LIN {X 0,Y 532.094,Z 203.208,A -85,B 0,C 180,E1 -4182.718,E2 -4182.718} C_VEL
LIN {X 0,Y 531.047,Z 203.336,A -85,B 0,C 180,E1 -4183.349,E2 -4183.349} C_VEL
LIN {X 0,Y 530.959,Z 203.344,A -85,B 0,C 180,E1 -4183.563,E2 -4183.563} C_VEL
LIN {X 0,Y 530.963,Z 203.345,A -85,B 0,C 180,E1 -4186.507,E2 -4186.507} C_VEL
LIN {X 0,Y 530.986,Z 203.345,A -85,B 0,C 180,E1 -4188.977,E2 -4188.977} C_VEL
LIN {X 0,Y 530.955,Z 203.343,A -85,B 0,C 180,E1 -4191.53,E2 -4191.53} C_VEL
LIN {X 0,Y 530.953,Z 203.348,A -85,B 0,C 180,E1 -4194.381,E2 -4194.381} C_VEL
LIN {X 0,Y 531.017,Z 203.34,A -85,B 0,C 180,E1 -4197.138,E2 -4197.138} C_VEL
LIN {X 0,Y 530.961,Z 203.352,A -85,B 0,C 180,E1 -4198.311,E2 -4198.311} C_VEL
LIN {X 0,Y 530.989,Z 212.149,A -85,B 0,C 180,E1 -4199.578,E2 -4199.578} C_VEL
LIN {X 0,Y 531.066,Z 222.092,A -85,B 0,C 180,E1 -4201.078,E2 -4201.078} C_VEL
LIN {X 0,Y 532.836,Z 233.019,A -85,B 0,C 180,E1 -4201.293,E2 -4201.293} C_VEL
LIN {X 0,Y 532.369,Z 329.637,A -85,B 0,C 180,E1 -4202.615,E2 -4202.615} C_VEL
LIN {X 0,Y 532.211,Z 343.265,A -85,B 0,C 180,E1 -4202.952,E2 -4202.952} C_VEL
LIN {X 0,Y 532.009,Z 355.388,A -85,B 0,C 180,E1 -4203.408,E2 -4203.408} C_VEL
LIN {X 0,Y 531.839,Z 368.214,A -85,B 0,C 180,E1 -4204.069,E2 -4204.069} C_VEL
LIN {X 0,Y 531.531,Z 378.711,A -85,B 0,C 180,E1 -4204.761,E2 -4204.761} C_VEL
LIN {X 0,Y 531.349,Z 388.715,A -85,B 0,C 180,E1 -4205.587,E2 -4205.587} C_VEL
LIN {X 0,Y 531.056,Z 398.766,A -85,B 0,C 180,E1 -4206.609,E2 -4206.609} C_VEL
LIN {X 0,Y 530.884,Z 407.591,A -85,B 0,C 180,E1 -4207.727,E2 -4207.727} C_VEL
LIN {X 0,Y 530.71,Z 414.712,A -85,B 0,C 180,E1 -4208.848,E2 -4208.848} C_VEL
LIN {X 0,Y 530.596,Z 421.185,A -85,B 0,C 180,E1 -4210.125,E2 -4210.125} C_VEL
LIN {X 0,Y 530.511,Z 426.324,A -85,B 0,C 180,E1 -4211.462,E2 -4211.462} C_VEL
LIN {X 0,Y 530.462,Z 429.415,A -85,B 0,C 180,E1 -4212.54,E2 -4212.54} C_VEL
LIN {X 0,Y 530.377,Z 431.976,A -85,B 0,C 180,E1 -4213.844,E2 -4213.844} C_VEL
LIN {X 0,Y 530.394,Z 433.447,A -85,B 0,C 180,E1 -4215.307,E2 -4215.307} C_VEL
LIN {X 0,Y 530.393,Z 433.621,A -85,B 0,C 180,E1 -4216.202,E2 -4216.202} C_VEL
LIN {X 0,Y 530.39,Z 433.323,A -85,B 0,C 180,E1 -4216.983,E2 -4216.983} C_VEL
LIN {X 0,Y 530.405,Z 432.632,A -85,B 0,C 180,E1 -4217.761,E2 -4217.761} C_VEL
LIN {X 0,Y 530.452,Z 431.3,A -85,B 0,C 180,E1 -4218.649,E2 -4218.649} C_VEL
LIN {X 0,Y 530.506,Z 427.984,A -85,B 0,C 180,E1 -4220.084,E2 -4220.084} C_VEL
LIN {X 0,Y 530.552,Z 424.156,A -85,B 0,C 180,E1 -4221.239,E2 -4221.239} C_VEL
LIN {X 0,Y 530.628,Z 419.211,A -85,B 0,C 180,E1 -4222.39,E2 -4222.39} C_VEL
LIN {X 0,Y 530.755,Z 412.935,A -85,B 0,C 180,E1 -4223.544,E2 -4223.544} C_VEL
LIN {X 0,Y 530.896,Z 405.219,A -85,B 0,C 180,E1 -4224.684,E2 -4224.684} C_VEL
LIN {X 0,Y 531.086,Z 397.332,A -85,B 0,C 180,E1 -4225.637,E2 -4225.637} C_VEL
LIN {X 0,Y 531.331,Z 387.768,A -85,B 0,C 180,E1 -4226.588,E2 -4226.588} C_VEL
LIN {X 0,Y 531.578,Z 377.06,A -85,B 0,C 180,E1 -4227.443,E2 -4227.443} C_VEL
LIN {X 0,Y 531.866,Z 365.041,A -85,B 0,C 180,E1 -4228.202,E2 -4228.202} C_VEL
LIN {X 0,Y 532.062,Z 353.262,A -85,B 0,C 180,E1 -4228.771,E2 -4228.771} C_VEL
LIN {X 0,Y 532.299,Z 339.567,A -85,B 0,C 180,E1 -4229.244,E2 -4229.244} C_VEL
LIN {X 0,Y 532.421,Z 326.575,A -85,B 0,C 180,E1 -4229.528,E2 -4229.528} C_VEL
LIN {X 0,Y 532.723,Z 231.859,A -85,B 0,C 180,E1 -4230.816,E2 -4230.816} C_VEL
LIN {X 0,Y 531.054,Z 222.286,A -85,B 0,C 180,E1 -4230.996,E2 -4230.996} C_VEL
LIN {X 0,Y 530.956,Z 203.717,A -85,B 0,C 180,E1 -4233.796,E2 -4233.796} C_VEL
LIN {X 0,Y 530.953,Z 203.352,A -85,B 0,C 180,E1 -4233.891,E2 -4233.891} C_VEL
LIN {X 0,Y 531.054,Z 203.332,A -85,B 0,C 180,E1 -4236.078,E2 -4236.078} C_VEL
LIN {X 0,Y 531.014,Z 203.342,A -85,B 0,C 180,E1 -4239.139,E2 -4239.139} C_VEL
LIN {X 0,Y 531.033,Z 203.334,A -85,B 0,C 180,E1 -4242.226,E2 -4242.226} C_VEL
LIN {X 0,Y 530.997,Z 203.344,A -85,B 0,C 180,E1 -4245.35,E2 -4245.35} C_VEL
LIN {X 0,Y 530.979,Z 203.342,A -85,B 0,C 180,E1 -4248.522,E2 -4248.522} C_VEL
LIN {X 0,Y 531.003,Z 203.344,A -85,B 0,C 180,E1 -4250.939,E2 -4250.939} C_VEL
LIN {X 0,Y 530.955,Z 203.344,A -85,B 0,C 180,E1 -4254.226,E2 -4254.226} C_VEL
LIN {X 0,Y 530.953,Z 203.35,A -85,B 0,C 180,E1 -4256.747,E2 -4256.747} C_VEL
LIN {X 0,Y 530.968,Z 203.344,A -85,B 0,C 180,E1 -4259.324,E2 -4259.324} C_VEL
LIN {X 0,Y 530.962,Z 203.344,A -85,B 0,C 180,E1 -4262.099,E2 -4262.099} C_VEL
LIN {X 0,Y 530.96,Z 203.349,A -85,B 0,C 180,E1 -4264.849,E2 -4264.849} C_VEL
LIN {X 0,Y 530.941,Z 203.345,A -85,B 0,C 180,E1 -4267.511,E2 -4267.511} C_VEL
LIN {X 0,Y 530.912,Z 203.355,A -85,B 0,C 180,E1 -4270.44,E2 -4270.44} C_VEL
LIN {X 0,Y 530.93,Z 203.347,A -85,B 0,C 180,E1 -4273.499,E2 -4273.499} C_VEL
LIN {X 0,Y 530.967,Z 203.343,A -85,B 0,C 180,E1 -4275.624,E2 -4275.624} C_VEL
LIN {X 0,Y 530.912,Z 203.353,A -85,B 0,C 180,E1 -4278.556,E2 -4278.556} C_VEL
LIN {X 0,Y 530.919,Z 203.35,A -85,B 0,C 180,E1 -4281.525,E2 -4281.525} C_VEL
LIN {X 0,Y 530.922,Z 203.352,A -85,B 0,C 180,E1 -4284.377,E2 -4284.377} C_VEL
LIN {X 0,Y 530.95,Z 203.344,A -85,B 0,C 180,E1 -4287.132,E2 -4287.132} C_VEL
LIN {X 0,Y 530.946,Z 203.351,A -85,B 0,C 180,E1 -4289.801,E2 -4289.801} C_VEL
LIN {X 0,Y 530.958,Z 203.345,A -85,B 0,C 180,E1 -4292.48,E2 -4292.48} C_VEL
LIN {X 0,Y 530.955,Z 203.349,A -85,B 0,C 180,E1 -4295.774,E2 -4295.774} C_VEL
LIN {X 0,Y 530.999,Z 203.34,A -85,B 0,C 180,E1 -4299.062,E2 -4299.062} C_VEL
LIN {X 0,Y 531.023,Z 203.373,A -85,B 0,C 180,E1 -4299.998,E2 -4299.998} C_VEL
LIN {X 0,Y 531.444,Z 208.695,A -85,B 0,C 180,E1 -4301.095,E2 -4301.095} C_VEL
LIN {X 0,Y 531.21,Z 222.508,A -85,B 0,C 180,E1 -4303.869,E2 -4303.869} C_VEL
LIN {X 0,Y 531.185,Z 223.727,A -85,B 0,C 180,E1 -4304.112,E2 -4304.112} C_VEL
LIN {X 0,Y 532.798,Z 232.98,A -85,B 0,C 180,E1 -4304.304,E2 -4304.304} C_VEL
LIN {X 0,Y 532.283,Z 330.71,A -85,B 0,C 180,E1 -4305.691,E2 -4305.691} C_VEL
LIN {X 0,Y 532.151,Z 344.492,A -85,B 0,C 180,E1 -4306.053,E2 -4306.053} C_VEL
LIN {X 0,Y 531.982,Z 356.812,A -85,B 0,C 180,E1 -4306.535,E2 -4306.535} C_VEL
LIN {X 0,Y 531.674,Z 369.545,A -85,B 0,C 180,E1 -4307.208,E2 -4307.208} C_VEL
LIN {X 0,Y 531.477,Z 380.023,A -85,B 0,C 180,E1 -4307.921,E2 -4307.921} C_VEL
LIN {X 0,Y 531.28,Z 389.834,A -85,B 0,C 180,E1 -4308.748,E2 -4308.748} C_VEL
LIN {X 0,Y 531.052,Z 399.176,A -85,B 0,C 180,E1 -4309.708,E2 -4309.708} C_VEL
LIN {X 0,Y 530.837,Z 408.2,A -85,B 0,C 180,E1 -4310.858,E2 -4310.858} C_VEL
LIN {X 0,Y 530.708,Z 415.384,A -85,B 0,C 180,E1 -4312.007,E2 -4312.007} C_VEL
LIN {X 0,Y 530.597,Z 421.13,A -85,B 0,C 180,E1 -4313.153,E2 -4313.153} C_VEL
LIN {X 0,Y 530.579,Z 425.659,A -85,B 0,C 180,E1 -4314.298,E2 -4314.298} C_VEL
LIN {X 0,Y 530.47,Z 429.1,A -85,B 0,C 180,E1 -4315.44,E2 -4315.44} C_VEL
LIN {X 0,Y 530.509,Z 432.156,A -85,B 0,C 180,E1 -4316.962,E2 -4316.962} C_VEL
LIN {X 0,Y 530.411,Z 433.041,A -85,B 0,C 180,E1 -4317.722,E2 -4317.722} C_VEL
LIN {X 0,Y 530.359,Z 433.646,A -85,B 0,C 180,E1 -4319.241,E2 -4319.241} C_VEL
LIN {X 0,Y 530.36,Z 433.356,A -85,B 0,C 180,E1 -4320,E2 -4320} C_VEL
LIN {X 0,Y 530.375,Z 431.556,A -85,B 0,C 180,E1 -4321.518,E2 -4321.518} C_VEL
LIN {X 0,Y 530.438,Z 430.066,A -85,B 0,C 180,E1 -4322.278,E2 -4322.278} C_VEL
LIN {X 0,Y 530.567,Z 426.982,A -85,B 0,C 180,E1 -4323.417,E2 -4323.417} C_VEL
LIN {X 0,Y 530.628,Z 422.844,A -85,B 0,C 180,E1 -4324.558,E2 -4324.558} C_VEL
LIN {X 0,Y 530.662,Z 417.53,A -85,B 0,C 180,E1 -4325.7,E2 -4325.7} C_VEL
LIN {X 0,Y 530.752,Z 411.655,A -85,B 0,C 180,E1 -4326.72,E2 -4326.72} C_VEL
LIN {X 0,Y 530.938,Z 404.064,A -85,B 0,C 180,E1 -4327.798,E2 -4327.798} C_VEL
LIN {X 0,Y 531.155,Z 395.87,A -85,B 0,C 180,E1 -4328.752,E2 -4328.752} C_VEL
LIN {X 0,Y 531.38,Z 385.827,A -85,B 0,C 180,E1 -4329.708,E2 -4329.708} C_VEL
LIN {X 0,Y 531.581,Z 374.406,A -85,B 0,C 180,E1 -4330.57,E2 -4330.57} C_VEL
LIN {X 0,Y 531.866,Z 363.178,A -85,B 0,C 180,E1 -4331.239,E2 -4331.239} C_VEL
LIN {X 0,Y 532.059,Z 351.412,A -85,B 0,C 180,E1 -4331.781,E2 -4331.781} C_VEL
LIN {X 0,Y 532.145,Z 337.987,A -85,B 0,C 180,E1 -4332.219,E2 -4332.219} C_VEL
LIN {X 0,Y 532.278,Z 325.431,A -85,B 0,C 180,E1 -4332.476,E2 -4332.476} C_VEL
LIN {X 0,Y 532.773,Z 233.014,A -85,B 0,C 180,E1 -4333.784,E2 -4333.784} C_VEL
LIN {X 0,Y 531.246,Z 224.418,A -85,B 0,C 180,E1 -4333.971,E2 -4333.971} C_VEL
LIN {X 0,Y 531.611,Z 210.036,A -85,B 0,C 180,E1 -4336.908,E2 -4336.908} C_VEL
LIN {X 0,Y 531.462,Z 205.781,A -85,B 0,C 180,E1 -4337.8,E2 -4337.8} C_VEL
LIN {X 0,Y 531.022,Z 203.343,A -85,B 0,C 180,E1 -4338.355,E2 -4338.355} C_VEL
LIN {X 0,Y 531.004,Z 203.342,A -85,B 0,C 180,E1 -4340.938,E2 -4340.938} C_VEL
LIN {X 0,Y 530.968,Z 203.349,A -85,B 0,C 180,E1 -4344.225,E2 -4344.225} C_VEL
LIN {X 0,Y 531.004,Z 203.342,A -85,B 0,C 180,E1 -4346.744,E2 -4346.744} C_VEL
LIN {X 0,Y 530.986,Z 203.34,A -85,B 0,C 180,E1 -4349.322,E2 -4349.322} C_VEL
LIN {X 0,Y 530.97,Z 203.348,A -85,B 0,C 180,E1 -4352.1,E2 -4352.1} C_VEL
LIN {X 0,Y 530.975,Z 203.342,A -85,B 0,C 180,E1 -4354.851,E2 -4354.851} C_VEL
LIN {X 0,Y 530.97,Z 203.342,A -85,B 0,C 180,E1 -4357.507,E2 -4357.507} C_VEL
LIN {X 0,Y 530.986,Z 203.344,A -85,B 0,C 180,E1 -4360.433,E2 -4360.433} C_VEL
LIN {X 0,Y 530.966,Z 203.342,A -85,B 0,C 180,E1 -4363.281,E2 -4363.281} C_VEL
LIN {X 0,Y 530.982,Z 203.342,A -85,B 0,C 180,E1 -4365.622,E2 -4365.622} C_VEL
LIN {X 0,Y 530.992,Z 203.341,A -85,B 0,C 180,E1 -4368.563,E2 -4368.563} C_VEL
LIN {X 0,Y 530.959,Z 203.345,A -85,B 0,C 180,E1 -4371.529,E2 -4371.529} C_VEL
LIN {X 0,Y 530.955,Z 203.347,A -85,B 0,C 180,E1 -4374.379,E2 -4374.379} C_VEL
LIN {X 0,Y 530.972,Z 203.343,A -85,B 0,C 180,E1 -4377.133,E2 -4377.133} C_VEL
LIN {X 0,Y 530.974,Z 203.352,A -85,B 0,C 180,E1 -4379.802,E2 -4379.802} C_VEL
LIN {X 0,Y 530.972,Z 203.346,A -85,B 0,C 180,E1 -4382.477,E2 -4382.477} C_VEL
LIN {X 0,Y 531.084,Z 203.525,A -85,B 0,C 180,E1 -4385.259,E2 -4385.259} C_VEL
LIN {X 0,Y 532.31,Z 210.932,A -85,B 0,C 180,E1 -4386.459,E2 -4386.459} C_VEL
LIN {X 0,Y 532.037,Z 227.094,A -85,B 0,C 180,E1 -4388.901,E2 -4388.901} C_VEL
LIN {X 0,Y 531.574,Z 249.168,A -85,B 0,C 180,E1 -4392.161,E2 -4392.161} C_VEL
LIN {X 0,Y 531.234,Z 269.092,A -85,B 0,C 180,E1 -4395.055,E2 -4395.055} C_VEL
LIN {X 0,Y 532.686,Z 280.104,A -85,B 0,C 180,E1 -4395.263,E2 -4395.263} C_VEL
LIN {X 0,Y 532.255,Z 376.467,A -85,B 0,C 180,E1 -4396.615,E2 -4396.615} C_VEL
LIN {X 0,Y 532.109,Z 389.547,A -85,B 0,C 180,E1 -4396.927,E2 -4396.927} C_VEL
LIN {X 0,Y 531.886,Z 402.741,A -85,B 0,C 180,E1 -4397.406,E2 -4397.406} C_VEL
LIN {X 0,Y 531.716,Z 414.517,A -85,B 0,C 180,E1 -4397.988,E2 -4397.988} C_VEL
LIN {X 0,Y 531.387,Z 426.388,A -85,B 0,C 180,E1 -4398.75,E2 -4398.75} C_VEL
LIN {X 0,Y 531.173,Z 437.085,A -85,B 0,C 180,E1 -4399.614,E2 -4399.614} C_VEL
LIN {X 0,Y 530.964,Z 445.824,A -85,B 0,C 180,E1 -4400.476,E2 -4400.476} C_VEL
LIN {X 0,Y 530.822,Z 453.873,A -85,B 0,C 180,E1 -4401.433,E2 -4401.433} C_VEL
LIN {X 0,Y 530.666,Z 461.728,A -85,B 0,C 180,E1 -4402.58,E2 -4402.58} C_VEL
LIN {X 0,Y 530.569,Z 468.927,A -85,B 0,C 180,E1 -4403.916,E2 -4403.916} C_VEL
LIN {X 0,Y 530.459,Z 473.721,A -85,B 0,C 180,E1 -4405.059,E2 -4405.059} C_VEL
LIN {X 0,Y 530.516,Z 477.39,A -85,B 0,C 180,E1 -4406.201,E2 -4406.201} C_VEL
LIN {X 0,Y 530.457,Z 479.283,A -85,B 0,C 180,E1 -4406.961,E2 -4406.961} C_VEL
LIN {X 0,Y 530.411,Z 480.695,A -85,B 0,C 180,E1 -4407.721,E2 -4407.721} C_VEL
LIN {X 0,Y 530.35,Z 482.317,A -85,B 0,C 180,E1 -4409.24,E2 -4409.24} C_VEL
LIN {X 0,Y 530.351,Z 482.541,A -85,B 0,C 180,E1 -4409.999,E2 -4409.999} C_VEL
LIN {X 0,Y 530.35,Z 482.326,A -85,B 0,C 180,E1 -4410.758,E2 -4410.758} C_VEL
LIN {X 0,Y 530.411,Z 480.716,A -85,B 0,C 180,E1 -4412.277,E2 -4412.277} C_VEL
LIN {X 0,Y 530.457,Z 479.309,A -85,B 0,C 180,E1 -4413.037,E2 -4413.037} C_VEL
LIN {X 0,Y 530.522,Z 476.355,A -85,B 0,C 180,E1 -4414.177,E2 -4414.177} C_VEL
LIN {X 0,Y 530.521,Z 472.347,A -85,B 0,C 180,E1 -4415.32,E2 -4415.32} C_VEL
LIN {X 0,Y 530.559,Z 466.754,A -85,B 0,C 180,E1 -4416.544,E2 -4416.544} C_VEL
LIN {X 0,Y 530.718,Z 459.417,A -85,B 0,C 180,E1 -4417.8,E2 -4417.8} C_VEL
LIN {X 0,Y 530.896,Z 451.031,A -85,B 0,C 180,E1 -4418.948,E2 -4418.948} C_VEL
LIN {X 0,Y 531.048,Z 442.399,A -85,B 0,C 180,E1 -4419.906,E2 -4419.906} C_VEL
LIN {X 0,Y 531.323,Z 431.749,A -85,B 0,C 180,E1 -4420.864,E2 -4420.864} C_VEL
LIN {X 0,Y 531.556,Z 420.954,A -85,B 0,C 180,E1 -4421.647,E2 -4421.647} C_VEL
LIN {X 0,Y 531.797,Z 409.531,A -85,B 0,C 180,E1 -4422.303,E2 -4422.303} C_VEL
LIN {X 0,Y 531.998,Z 397.424,A -85,B 0,C 180,E1 -4422.832,E2 -4422.832} C_VEL
LIN {X 0,Y 532.207,Z 384.319,A -85,B 0,C 180,E1 -4423.239,E2 -4423.239} C_VEL
LIN {X 0,Y 532.37,Z 370.239,A -85,B 0,C 180,E1 -4423.502,E2 -4423.502} C_VEL
LIN {X 0,Y 532.56,Z 278.274,A -85,B 0,C 180,E1 -4424.775,E2 -4424.775} C_VEL
LIN {X 0,Y 531.29,Z 269.694,A -85,B 0,C 180,E1 -4424.94,E2 -4424.94} C_VEL
LIN {X 0,Y 531.727,Z 248.102,A -85,B 0,C 180,E1 -4428.118,E2 -4428.118} C_VEL
LIN {X 0,Y 532.186,Z 226.695,A -85,B 0,C 180,E1 -4431.294,E2 -4431.294} C_VEL
LIN {X 0,Y 532.557,Z 211.959,A -85,B 0,C 180,E1 -4433.527,E2 -4433.527} C_VEL
LIN {X 0,Y 531.027,Z 203.339,A -85,B 0,C 180,E1 -4434.951,E2 -4434.951} C_VEL
LIN {X 0,Y 531.006,Z 203.341,A -85,B 0,C 180,E1 -4437.595,E2 -4437.595} C_VEL
LIN {X 0,Y 530.971,Z 203.342,A -85,B 0,C 180,E1 -4440.644,E2 -4440.644} C_VEL
LIN {X 0,Y 530.983,Z 203.336,A -85,B 0,C 180,E1 -4443.772,E2 -4443.772} C_VEL
LIN {X 0,Y 530.946,Z 203.344,A -85,B 0,C 180,E1 -4446.558,E2 -4446.558} C_VEL
LIN {X 0,Y 530.966,Z 203.343,A -85,B 0,C 180,E1 -4449.444,E2 -4449.444} C_VEL
LIN {X 0,Y 530.958,Z 203.341,A -85,B 0,C 180,E1 -4452.457,E2 -4452.457} C_VEL
LIN {X 0,Y 530.961,Z 203.348,A -85,B 0,C 180,E1 -4455.45,E2 -4455.45} C_VEL
LIN {X 0,Y 530.957,Z 203.338,A -85,B 0,C 180,E1 -4458.561,E2 -4458.561} C_VEL
LIN {X 0,Y 530.946,Z 203.349,A -85,B 0,C 180,E1 -4461.528,E2 -4461.528} C_VEL
LIN {X 0,Y 530.946,Z 203.337,A -85,B 0,C 180,E1 -4464.379,E2 -4464.379} C_VEL
LIN {X 0,Y 530.956,Z 203.348,A -85,B 0,C 180,E1 -4467.133,E2 -4467.133} C_VEL
LIN {X 0,Y 530.937,Z 203.339,A -85,B 0,C 180,E1 -4469.801,E2 -4469.801} C_VEL
LIN {X 0,Y 530.953,Z 203.34,A -85,B 0,C 180,E1 -4472.478,E2 -4472.478} C_VEL
LIN {X 0,Y 530.936,Z 203.352,A -85,B 0,C 180,E1 -4474.939,E2 -4474.939} C_VEL
LIN {X 0,Y 530.966,Z 203.332,A -85,B 0,C 180,E1 -4477.898,E2 -4477.898} C_VEL
LIN {X 0,Y 530.953,Z 203.346,A -85,B 0,C 180,E1 -4480.676,E2 -4480.676} C_VEL
LIN {X 0,Y 530.942,Z 203.346,A -85,B 0,C 180,E1 -4483.07,E2 -4483.07} C_VEL
LIN {X 0,Y 530.987,Z 203.331,A -85,B 0,C 180,E1 -4485.435,E2 -4485.435} C_VEL
LIN {X 0,Y 531.021,Z 203.339,A -85,B 0,C 180,E1 -4488.549,E2 -4488.549} C_VEL
LIN {X 0,Y 531.019,Z 203.334,A -85,B 0,C 180,E1 -4491.629,E2 -4491.629} C_VEL
LIN {X 0,Y 531.076,Z 203.326,A -85,B 0,C 180,E1 -4494.685,E2 -4494.685} C_VEL
LIN {X 0,Y 531.12,Z 203.321,A -85,B 0,C 180,E1 -4497.725,E2 -4497.725} C_VEL
LIN {X 0,Y 531.14,Z 203.317,A -85,B 0,C 180,E1 -4500.758,E2 -4500.758} C_VEL
LIN {X 0,Y 531.08,Z 203.319,A -85,B 0,C 180,E1 -4503.034,E2 -4503.034} C_VEL
LIN {X 0,Y 531.068,Z 203.335,A -85,B 0,C 180,E1 -4506.077,E2 -4506.077} C_VEL
LIN {X 0,Y 531.042,Z 203.331,A -85,B 0,C 180,E1 -4508.371,E2 -4508.371} C_VEL
LIN {X 0,Y 531.043,Z 203.33,A -85,B 0,C 180,E1 -4511.672,E2 -4511.672} C_VEL
LIN {X 0,Y 531.023,Z 203.333,A -85,B 0,C 180,E1 -4514.956,E2 -4514.956} C_VEL
LIN {X 0,Y 530.973,Z 203.342,A -85,B 0,C 180,E1 -4517.724,E2 -4517.724} C_VEL
LIN {X 0,Y 531.017,Z 203.337,A -85,B 0,C 180,E1 -4520.128,E2 -4520.128} C_VEL
LIN {X 0,Y 530.957,Z 203.346,A -85,B 0,C 180,E1 -4523.397,E2 -4523.397} C_VEL
LIN {X 0,Y 531.006,Z 203.34,A -85,B 0,C 180,E1 -4525.898,E2 -4525.898} C_VEL
LIN {X 0,Y 530.966,Z 203.339,A -85,B 0,C 180,E1 -4528.458,E2 -4528.458} C_VEL
LIN {X 0,Y 530.952,Z 203.346,A -85,B 0,C 180,E1 -4531.08,E2 -4531.08} C_VEL
LIN {X 0,Y 530.984,Z 203.339,A -85,B 0,C 180,E1 -4533.773,E2 -4533.773} C_VEL
LIN {X 0,Y 530.962,Z 203.344,A -85,B 0,C 180,E1 -4536.558,E2 -4536.558} C_VEL
LIN {X 0,Y 530.978,Z 203.341,A -85,B 0,C 180,E1 -4539.855,E2 -4539.855} C_VEL
LIN {X 0,Y 530.975,Z 203.34,A -85,B 0,C 180,E1 -4542.458,E2 -4542.458} C_VEL
LIN {X 0,Y 530.959,Z 203.344,A -85,B 0,C 180,E1 -4543.563,E2 -4543.563} C_VEL
LIN {X 0,Y 530.287,Z 203.427,A -85,B 0,C 180,E1 -4544.197,E2 -4544.197} C_VEL
LIN {X 0,Y 527.44,Z 203.789,A -85,B 0,C 180,E1 -4545.225,E2 -4545.225} C_VEL
LIN {X 0,Y 525.036,Z 204.093,A -85,B 0,C 180,E1 -4546.054,E2 -4546.054} C_VEL
LIN {X 0,Y 524.003,Z 204.218,A -85,B 0,C 180,E1 -4546.693,E2 -4546.693} C_VEL
LIN {X 0,Y 523.917,Z 204.226,A -85,B 0,C 180,E1 -4546.91,E2 -4546.91} C_VEL
LIN {X 0,Y 523.946,Z 204.215,A -85,B 0,C 180,E1 -4549.922,E2 -4549.922} C_VEL
LIN {X 0,Y 523.906,Z 204.228,A -85,B 0,C 180,E1 -4552.869,E2 -4552.869} C_VEL
LIN {X 0,Y 523.936,Z 204.219,A -85,B 0,C 180,E1 -4555.711,E2 -4555.711} C_VEL
LIN {X 0,Y 523.93,Z 204.299,A -85,B 0,C 180,E1 -4558.331,E2 -4558.331} C_VEL
LIN {X 0,Y 523.983,Z 211.815,A -85,B 0,C 180,E1 -4559.359,E2 -4559.359} C_VEL
LIN {X 0,Y 524.042,Z 222.175,A -85,B 0,C 180,E1 -4560.885,E2 -4560.885} C_VEL
LIN {X 0,Y 525.988,Z 234.235,A -85,B 0,C 180,E1 -4561.111,E2 -4561.111} C_VEL
LIN {X 0,Y 525.492,Z 330.171,A -85,B 0,C 180,E1 -4562.442,E2 -4562.442} C_VEL
LIN {X 0,Y 525.3,Z 343.701,A -85,B 0,C 180,E1 -4562.782,E2 -4562.782} C_VEL
LIN {X 0,Y 525.099,Z 356.012,A -85,B 0,C 180,E1 -4563.255,E2 -4563.255} C_VEL
LIN {X 0,Y 524.888,Z 368.893,A -85,B 0,C 180,E1 -4563.93,E2 -4563.93} C_VEL
LIN {X 0,Y 524.548,Z 380.423,A -85,B 0,C 180,E1 -4564.719,E2 -4564.719} C_VEL
LIN {X 0,Y 524.318,Z 390.973,A -85,B 0,C 180,E1 -4565.631,E2 -4565.631} C_VEL
LIN {X 0,Y 524.059,Z 399.12,A -85,B 0,C 180,E1 -4566.487,E2 -4566.487} C_VEL
LIN {X 0,Y 523.882,Z 407.051,A -85,B 0,C 180,E1 -4567.493,E2 -4567.493} C_VEL
LIN {X 0,Y 523.651,Z 415.051,A -85,B 0,C 180,E1 -4568.755,E2 -4568.755} C_VEL
LIN {X 0,Y 523.528,Z 421.307,A -85,B 0,C 180,E1 -4570.003,E2 -4570.003} C_VEL
LIN {X 0,Y 523.46,Z 425.994,A -85,B 0,C 180,E1 -4571.203,E2 -4571.203} C_VEL
LIN {X 0,Y 523.391,Z 429.599,A -85,B 0,C 180,E1 -4572.437,E2 -4572.437} C_VEL
LIN {X 0,Y 523.294,Z 432.008,A -85,B 0,C 180,E1 -4573.619,E2 -4573.619} C_VEL
LIN {X 0,Y 523.259,Z 433.067,A -85,B 0,C 180,E1 -4574.419,E2 -4574.419} C_VEL
LIN {X 0,Y 523.307,Z 433.722,A -85,B 0,C 180,E1 -4575.232,E2 -4575.232} C_VEL
LIN {X 0,Y 523.304,Z 433.959,A -85,B 0,C 180,E1 -4576.012,E2 -4576.012} C_VEL
LIN {X 0,Y 523.292,Z 433.753,A -85,B 0,C 180,E1 -4576.803,E2 -4576.803} C_VEL
LIN {X 0,Y 523.354,Z 432.131,A -85,B 0,C 180,E1 -4578.38,E2 -4578.38} C_VEL
LIN {X 0,Y 523.36,Z 430.693,A -85,B 0,C 180,E1 -4579.165,E2 -4579.165} C_VEL
LIN {X 0,Y 523.44,Z 427.714,A -85,B 0,C 180,E1 -4580.339,E2 -4580.339} C_VEL
LIN {X 0,Y 523.498,Z 423.695,A -85,B 0,C 180,E1 -4581.509,E2 -4581.509} C_VEL
LIN {X 0,Y 523.569,Z 418.529,A -85,B 0,C 180,E1 -4582.675,E2 -4582.675} C_VEL
LIN {X 0,Y 523.736,Z 412.052,A -85,B 0,C 180,E1 -4583.838,E2 -4583.838} C_VEL
LIN {X 0,Y 523.939,Z 404.041,A -85,B 0,C 180,E1 -4584.999,E2 -4584.999} C_VEL
LIN {X 0,Y 524.148,Z 395.834,A -85,B 0,C 180,E1 -4585.964,E2 -4585.964} C_VEL
LIN {X 0,Y 524.411,Z 385.787,A -85,B 0,C 180,E1 -4586.928,E2 -4586.928} C_VEL
LIN {X 0,Y 524.719,Z 374.568,A -85,B 0,C 180,E1 -4587.794,E2 -4587.794} C_VEL
LIN {X 0,Y 524.973,Z 363.447,A -85,B 0,C 180,E1 -4588.467,E2 -4588.467} C_VEL
LIN {X 0,Y 525.198,Z 351.022,A -85,B 0,C 180,E1 -4589.042,E2 -4589.042} C_VEL
LIN {X 0,Y 525.43,Z 338.795,A -85,B 0,C 180,E1 -4589.45,E2 -4589.45} C_VEL
LIN {X 0,Y 525.546,Z 324.827,A -85,B 0,C 180,E1 -4589.737,E2 -4589.737} C_VEL
LIN {X 0,Y 525.955,Z 233.233,A -85,B 0,C 180,E1 -4590.994,E2 -4590.994} C_VEL
LIN {X 0,Y 524.067,Z 222.052,A -85,B 0,C 180,E1 -4591.226,E2 -4591.226} C_VEL
LIN {X 0,Y 523.909,Z 204.229,A -85,B 0,C 180,E1 -4593.847,E2 -4593.847} C_VEL
LIN {X 0,Y 524.02,Z 204.208,A -85,B 0,C 180,E1 -4596.16,E2 -4596.16} C_VEL
LIN {X 0,Y 523.99,Z 204.211,A -85,B 0,C 180,E1 -4598.485,E2 -4598.485} C_VEL
LIN {X 0,Y 524.004,Z 204.212,A -85,B 0,C 180,E1 -4601.737,E2 -4601.737} C_VEL
LIN {X 0,Y 523.99,Z 204.218,A -85,B 0,C 180,E1 -4605.048,E2 -4605.048} C_VEL
LIN {X 0,Y 523.951,Z 204.216,A -85,B 0,C 180,E1 -4607.97,E2 -4607.97} C_VEL
LIN {X 0,Y 523.964,Z 204.216,A -85,B 0,C 180,E1 -4610.411,E2 -4610.411} C_VEL
LIN {X 0,Y 523.914,Z 204.227,A -85,B 0,C 180,E1 -4612.894,E2 -4612.894} C_VEL
LIN {X 0,Y 523.901,Z 204.225,A -85,B 0,C 180,E1 -4615.422,E2 -4615.422} C_VEL
LIN {X 0,Y 523.912,Z 204.221,A -85,B 0,C 180,E1 -4618.003,E2 -4618.003} C_VEL
LIN {X 0,Y 523.916,Z 204.226,A -85,B 0,C 180,E1 -4620.848,E2 -4620.848} C_VEL
LIN {X 0,Y 523.93,Z 204.219,A -85,B 0,C 180,E1 -4623.729,E2 -4623.729} C_VEL
LIN {X 0,Y 523.884,Z 204.231,A -85,B 0,C 180,E1 -4626.398,E2 -4626.398} C_VEL
LIN {X 0,Y 523.901,Z 204.224,A -85,B 0,C 180,E1 -4629.087,E2 -4629.087} C_VEL
LIN {X 0,Y 523.879,Z 204.231,A -85,B 0,C 180,E1 -4632.451,E2 -4632.451} C_VEL
LIN {X 0,Y 523.937,Z 204.218,A -85,B 0,C 180,E1 -4635.312,E2 -4635.312} C_VEL
LIN {X 0,Y 523.881,Z 204.228,A -85,B 0,C 180,E1 -4638.7,E2 -4638.7} C_VEL
LIN {X 0,Y 523.873,Z 204.231,A -85,B 0,C 180,E1 -4641.894,E2 -4641.894} C_VEL
LIN {X 0,Y 523.891,Z 204.224,A -85,B 0,C 180,E1 -4644.918,E2 -4644.918} C_VEL
LIN {X 0,Y 523.904,Z 204.227,A -85,B 0,C 180,E1 -4647.686,E2 -4647.686} C_VEL
LIN {X 0,Y 523.878,Z 204.23,A -85,B 0,C 180,E1 -4650.24,E2 -4650.24} C_VEL
LIN {X 0,Y 523.895,Z 204.223,A -85,B 0,C 180,E1 -4652.863,E2 -4652.863} C_VEL
LIN {X 0,Y 523.938,Z 204.223,A -85,B 0,C 180,E1 -4655.804,E2 -4655.804} C_VEL
LIN {X 0,Y 523.948,Z 204.218,A -85,B 0,C 180,E1 -4658.766,E2 -4658.766} C_VEL
LIN {X 0,Y 524.017,Z 204.308,A -85,B 0,C 180,E1 -4659.888,E2 -4659.888} C_VEL
LIN {X 0,Y 524.433,Z 210.793,A -85,B 0,C 180,E1 -4661.238,E2 -4661.238} C_VEL
LIN {X 0,Y 524.196,Z 224.018,A -85,B 0,C 180,E1 -4663.917,E2 -4663.917} C_VEL
LIN {X 0,Y 525.931,Z 233.245,A -85,B 0,C 180,E1 -4664.11,E2 -4664.11} C_VEL
LIN {X 0,Y 525.377,Z 330.705,A -85,B 0,C 180,E1 -4665.523,E2 -4665.523} C_VEL
LIN {X 0,Y 525.211,Z 344.557,A -85,B 0,C 180,E1 -4665.889,E2 -4665.889} C_VEL
LIN {X 0,Y 525.053,Z 356.441,A -85,B 0,C 180,E1 -4666.354,E2 -4666.354} C_VEL
LIN {X 0,Y 524.786,Z 367.723,A -85,B 0,C 180,E1 -4666.939,E2 -4666.939} C_VEL
LIN {X 0,Y 524.54,Z 379.205,A -85,B 0,C 180,E1 -4667.706,E2 -4667.706} C_VEL
LIN {X 0,Y 524.294,Z 389.83,A -85,B 0,C 180,E1 -4668.596,E2 -4668.596} C_VEL
LIN {X 0,Y 524.038,Z 399.225,A -85,B 0,C 180,E1 -4669.569,E2 -4669.569} C_VEL
LIN {X 0,Y 523.807,Z 408.293,A -85,B 0,C 180,E1 -4670.734,E2 -4670.734} C_VEL
LIN {X 0,Y 523.648,Z 415.563,A -85,B 0,C 180,E1 -4671.899,E2 -4671.899} C_VEL
LIN {X 0,Y 523.552,Z 421.346,A -85,B 0,C 180,E1 -4673.061,E2 -4673.061} C_VEL
LIN {X 0,Y 523.514,Z 425.906,A -85,B 0,C 180,E1 -4674.221,E2 -4674.221} C_VEL
LIN {X 0,Y 523.378,Z 429.374,A -85,B 0,C 180,E1 -4675.379,E2 -4675.379} C_VEL
LIN {X 0,Y 523.443,Z 432.443,A -85,B 0,C 180,E1 -4676.921,E2 -4676.921} C_VEL
LIN {X 0,Y 523.336,Z 433.352,A -85,B 0,C 180,E1 -4677.691,E2 -4677.691} C_VEL
LIN {X 0,Y 523.267,Z 433.976,A -85,B 0,C 180,E1 -4679.23,E2 -4679.23} C_VEL
LIN {X 0,Y 523.268,Z 433.689,A -85,B 0,C 180,E1 -4680,E2 -4680} C_VEL
LIN {X 0,Y 523.288,Z 431.914,A -85,B 0,C 180,E1 -4681.539,E2 -4681.539} C_VEL
LIN {X 0,Y 523.362,Z 430.407,A -85,B 0,C 180,E1 -4682.309,E2 -4682.309} C_VEL
LIN {X 0,Y 523.5,Z 427.324,A -85,B 0,C 180,E1 -4683.463,E2 -4683.463} C_VEL
LIN {X 0,Y 523.57,Z 423.184,A -85,B 0,C 180,E1 -4684.619,E2 -4684.619} C_VEL
LIN {X 0,Y 523.616,Z 417.867,A -85,B 0,C 180,E1 -4685.777,E2 -4685.777} C_VEL
LIN {X 0,Y 523.742,Z 411.19,A -85,B 0,C 180,E1 -4686.936,E2 -4686.936} C_VEL
LIN {X 0,Y 523.932,Z 402.896,A -85,B 0,C 180,E1 -4688.097,E2 -4688.097} C_VEL
LIN {X 0,Y 524.186,Z 394.326,A -85,B 0,C 180,E1 -4689.064,E2 -4689.064} C_VEL
LIN {X 0,Y 524.42,Z 383.738,A -85,B 0,C 180,E1 -4690.033,E2 -4690.033} C_VEL
LIN {X 0,Y 524.684,Z 373.209,A -85,B 0,C 180,E1 -4690.808,E2 -4690.808} C_VEL
LIN {X 0,Y 524.939,Z 361.492,A -85,B 0,C 180,E1 -4691.487,E2 -4691.487} C_VEL
LIN {X 0,Y 525.175,Z 349.303,A -85,B 0,C 180,E1 -4692.02,E2 -4692.02} C_VEL
LIN {X 0,Y 525.243,Z 336.911,A -85,B 0,C 180,E1 -4692.411,E2 -4692.411} C_VEL
LIN {X 0,Y 525.341,Z 324.553,A -85,B 0,C 180,E1 -4692.654,E2 -4692.654} C_VEL
LIN {X 0,Y 525.918,Z 233.916,A -85,B 0,C 180,E1 -4693.968,E2 -4693.968} C_VEL
LIN {X 0,Y 524.288,Z 224.889,A -85,B 0,C 180,E1 -4694.16,E2 -4694.16} C_VEL
LIN {X 0,Y 524.61,Z 212.417,A -85,B 0,C 180,E1 -4696.74,E2 -4696.74} C_VEL
LIN {X 0,Y 524.446,Z 206.7,A -85,B 0,C 180,E1 -4697.952,E2 -4697.952} C_VEL
LIN {X 0,Y 523.967,Z 204.221,A -85,B 0,C 180,E1 -4698.525,E2 -4698.525} C_VEL
LIN {X 0,Y 523.951,Z 204.219,A -85,B 0,C 180,E1 -4701.233,E2 -4701.233} C_VEL
LIN {X 0,Y 523.927,Z 204.226,A -85,B 0,C 180,E1 -4704.572,E2 -4704.572} C_VEL
LIN {X 0,Y 523.953,Z 204.217,A -85,B 0,C 180,E1 -4707.133,E2 -4707.133} C_VEL
LIN {X 0,Y 523.943,Z 204.219,A -85,B 0,C 180,E1 -4709.756,E2 -4709.756} C_VEL
LIN {X 0,Y 523.938,Z 204.224,A -85,B 0,C 180,E1 -4712.449,E2 -4712.449} C_VEL
LIN {X 0,Y 523.925,Z 204.219,A -85,B 0,C 180,E1 -4715.226,E2 -4715.226} C_VEL
LIN {X 0,Y 523.92,Z 204.226,A -85,B 0,C 180,E1 -4718.101,E2 -4718.101} C_VEL
LIN {X 0,Y 523.944,Z 204.216,A -85,B 0,C 180,E1 -4721.092,E2 -4721.092} C_VEL
LIN {X 0,Y 523.936,Z 204.225,A -85,B 0,C 180,E1 -4724.228,E2 -4724.228} C_VEL
LIN {X 0,Y 523.906,Z 204.222,A -85,B 0,C 180,E1 -4726.831,E2 -4726.831} C_VEL
LIN {X 0,Y 523.939,Z 204.218,A -85,B 0,C 180,E1 -4728.907,E2 -4728.907} C_VEL
LIN {X 0,Y 523.918,Z 204.227,A -85,B 0,C 180,E1 -4731.897,E2 -4731.897} C_VEL
LIN {X 0,Y 523.928,Z 204.219,A -85,B 0,C 180,E1 -4734.911,E2 -4734.911} C_VEL
LIN {X 0,Y 523.94,Z 204.225,A -85,B 0,C 180,E1 -4737.679,E2 -4737.679} C_VEL
LIN {X 0,Y 523.958,Z 204.22,A -85,B 0,C 180,E1 -4740.676,E2 -4740.676} C_VEL
LIN {X 0,Y 523.936,Z 204.225,A -85,B 0,C 180,E1 -4743.726,E2 -4743.726} C_VEL
LIN {X 0,Y 524.006,Z 204.355,A -85,B 0,C 180,E1 -4745.061,E2 -4745.061} C_VEL
LIN {X 0,Y 525.366,Z 212.042,A -85,B 0,C 180,E1 -4746.338,E2 -4746.338} C_VEL
LIN {X 0,Y 525.108,Z 226.765,A -85,B 0,C 180,E1 -4748.609,E2 -4748.609} C_VEL
LIN {X 0,Y 524.559,Z 249.704,A -85,B 0,C 180,E1 -4752.051,E2 -4752.051} C_VEL
LIN {X 0,Y 524.228,Z 268.716,A -85,B 0,C 180,E1 -4754.854,E2 -4754.854} C_VEL
LIN {X 0,Y 525.829,Z 281.219,A -85,B 0,C 180,E1 -4755.09,E2 -4755.09} C_VEL
LIN {X 0,Y 525.297,Z 377.513,A -85,B 0,C 180,E1 -4756.483,E2 -4756.483} C_VEL
LIN {X 0,Y 525.087,Z 390.74,A -85,B 0,C 180,E1 -4756.823,E2 -4756.823} C_VEL
LIN {X 0,Y 524.857,Z 404.088,A -85,B 0,C 180,E1 -4757.333,E2 -4757.333} C_VEL
LIN {X 0,Y 524.664,Z 415.36,A -85,B 0,C 180,E1 -4757.92,E2 -4757.92} C_VEL
LIN {X 0,Y 524.333,Z 427.023,A -85,B 0,C 180,E1 -4758.694,E2 -4758.694} C_VEL
LIN {X 0,Y 524.124,Z 437.573,A -85,B 0,C 180,E1 -4759.57,E2 -4759.57} C_VEL
LIN {X 0,Y 523.875,Z 447.029,A -85,B 0,C 180,E1 -4760.54,E2 -4760.54} C_VEL
LIN {X 0,Y 523.682,Z 456.176,A -85,B 0,C 180,E1 -4761.704,E2 -4761.704} C_VEL
LIN {X 0,Y 523.57,Z 463.553,A -85,B 0,C 180,E1 -4762.867,E2 -4762.867} C_VEL
LIN {X 0,Y 523.467,Z 468.512,A -85,B 0,C 180,E1 -4763.833,E2 -4763.833} C_VEL
LIN {X 0,Y 523.383,Z 473.334,A -85,B 0,C 180,E1 -4764.992,E2 -4764.992} C_VEL
LIN {X 0,Y 523.443,Z 477.026,A -85,B 0,C 180,E1 -4766.15,E2 -4766.15} C_VEL
LIN {X 0,Y 523.368,Z 478.93,A -85,B 0,C 180,E1 -4766.92,E2 -4766.92} C_VEL
LIN {X 0,Y 523.335,Z 480.353,A -85,B 0,C 180,E1 -4767.69,E2 -4767.69} C_VEL
LIN {X 0,Y 523.258,Z 481.988,A -85,B 0,C 180,E1 -4769.23,E2 -4769.23} C_VEL
LIN {X 0,Y 523.259,Z 482.216,A -85,B 0,C 180,E1 -4769.999,E2 -4769.999} C_VEL
LIN {X 0,Y 523.257,Z 482.001,A -85,B 0,C 180,E1 -4770.769,E2 -4770.769} C_VEL
LIN {X 0,Y 523.335,Z 480.389,A -85,B 0,C 180,E1 -4772.308,E2 -4772.308} C_VEL
LIN {X 0,Y 523.367,Z 478.976,A -85,B 0,C 180,E1 -4773.078,E2 -4773.078} C_VEL
LIN {X 0,Y 523.423,Z 476.012,A -85,B 0,C 180,E1 -4774.234,E2 -4774.234} C_VEL
LIN {X 0,Y 523.455,Z 471.99,A -85,B 0,C 180,E1 -4775.392,E2 -4775.392} C_VEL
LIN {X 0,Y 523.509,Z 465.824,A -85,B 0,C 180,E1 -4776.738,E2 -4776.738} C_VEL
LIN {X 0,Y 523.655,Z 459.012,A -85,B 0,C 180,E1 -4777.906,E2 -4777.906} C_VEL
LIN {X 0,Y 523.831,Z 450.593,A -85,B 0,C 180,E1 -4779.069,E2 -4779.069} C_VEL
LIN {X 0,Y 523.998,Z 441.918,A -85,B 0,C 180,E1 -4780.04,E2 -4780.04} C_VEL
LIN {X 0,Y 524.325,Z 431.23,A -85,B 0,C 180,E1 -4781.011,E2 -4781.011} C_VEL
LIN {X 0,Y 524.511,Z 419.718,A -85,B 0,C 180,E1 -4781.85,E2 -4781.85} C_VEL
LIN {X 0,Y 524.805,Z 407.855,A -85,B 0,C 180,E1 -4782.519,E2 -4782.519} C_VEL
LIN {X 0,Y 525.061,Z 395.352,A -85,B 0,C 180,E1 -4783.053,E2 -4783.053} C_VEL
LIN {X 0,Y 525.315,Z 382.39,A -85,B 0,C 180,E1 -4783.441,E2 -4783.441} C_VEL
LIN {X 0,Y 525.481,Z 365.462,A -85,B 0,C 180,E1 -4783.732,E2 -4783.732} C_VEL
LIN {X 0,Y 525.729,Z 279.233,A -85,B 0,C 180,E1 -4784.953,E2 -4784.953} C_VEL
LIN {X 0,Y 524.278,Z 269.273,A -85,B 0,C 180,E1 -4785.166,E2 -4785.166} C_VEL
LIN {X 0,Y 524.738,Z 248.293,A -85,B 0,C 180,E1 -4788.304,E2 -4788.304} C_VEL
LIN {X 0,Y 525.271,Z 226.468,A -85,B 0,C 180,E1 -4791.588,E2 -4791.588} C_VEL
LIN {X 0,Y 525.627,Z 213.111,A -85,B 0,C 180,E1 -4793.647,E2 -4793.647} C_VEL
LIN {X 0,Y 524.005,Z 204.214,A -85,B 0,C 180,E1 -4795.149,E2 -4795.149} C_VEL
LIN {X 0,Y 523.954,Z 204.223,A -85,B 0,C 180,E1 -4797.999,E2 -4797.999} C_VEL
LIN {X 0,Y 523.941,Z 204.217,A -85,B 0,C 180,E1 -4800.854,E2 -4800.854} C_VEL
LIN {X 0,Y 523.955,Z 204.211,A -85,B 0,C 180,E1 -4803.733,E2 -4803.733} C_VEL
LIN {X 0,Y 523.894,Z 204.224,A -85,B 0,C 180,E1 -4806.4,E2 -4806.4} C_VEL
LIN {X 0,Y 523.908,Z 204.219,A -85,B 0,C 180,E1 -4809.085,E2 -4809.085} C_VEL
LIN {X 0,Y 523.934,Z 204.218,A -85,B 0,C 180,E1 -4812.119,E2 -4812.119} C_VEL
LIN {X 0,Y 523.932,Z 204.222,A -85,B 0,C 180,E1 -4815.31,E2 -4815.31} C_VEL
LIN {X 0,Y 523.917,Z 204.215,A -85,B 0,C 180,E1 -4818.693,E2 -4818.693} C_VEL
LIN {X 0,Y 523.906,Z 204.221,A -85,B 0,C 180,E1 -4821.897,E2 -4821.897} C_VEL
LIN {X 0,Y 523.916,Z 204.216,A -85,B 0,C 180,E1 -4824.911,E2 -4824.911} C_VEL
LIN {X 0,Y 523.922,Z 204.219,A -85,B 0,C 180,E1 -4827.68,E2 -4827.68} C_VEL
LIN {X 0,Y 523.926,Z 204.214,A -85,B 0,C 180,E1 -4830.68,E2 -4830.68} C_VEL
LIN {X 0,Y 523.891,Z 204.221,A -85,B 0,C 180,E1 -4833.724,E2 -4833.724} C_VEL
LIN {X 0,Y 523.897,Z 204.219,A -85,B 0,C 180,E1 -4836.269,E2 -4836.269} C_VEL
LIN {X 0,Y 523.92,Z 204.216,A -85,B 0,C 180,E1 -4838.766,E2 -4838.766} C_VEL
LIN {X 0,Y 523.917,Z 204.221,A -85,B 0,C 180,E1 -4841.22,E2 -4841.22} C_VEL
LIN {X 0,Y 523.879,Z 204.221,A -85,B 0,C 180,E1 -4843.637,E2 -4843.637} C_VEL
LIN {X 0,Y 523.898,Z 204.214,A -85,B 0,C 180,E1 -4846.027,E2 -4846.027} C_VEL
LIN {X 0,Y 524.004,Z 204.21,A -85,B 0,C 180,E1 -4848.394,E2 -4848.394} C_VEL
LIN {X 0,Y 523.972,Z 204.211,A -85,B 0,C 180,E1 -4851.516,E2 -4851.516} C_VEL
LIN {X 0,Y 524.021,Z 204.204,A -85,B 0,C 180,E1 -4854.613,E2 -4854.613} C_VEL
LIN {X 0,Y 524.093,Z 204.196,A -85,B 0,C 180,E1 -4857.695,E2 -4857.695} C_VEL
LIN {X 0,Y 524.111,Z 204.192,A -85,B 0,C 180,E1 -4860.769,E2 -4860.769} C_VEL
LIN {X 0,Y 524.02,Z 204.198,A -85,B 0,C 180,E1 -4863.075,E2 -4863.075} C_VEL
LIN {X 0,Y 524.032,Z 204.211,A -85,B 0,C 180,E1 -4866.159,E2 -4866.159} C_VEL
LIN {X 0,Y 523.99,Z 204.208,A -85,B 0,C 180,E1 -4868.484,E2 -4868.484} C_VEL
LIN {X 0,Y 523.994,Z 204.209,A -85,B 0,C 180,E1 -4871.739,E2 -4871.739} C_VEL
LIN {X 0,Y 523.985,Z 204.21,A -85,B 0,C 180,E1 -4875.053,E2 -4875.053} C_VEL
LIN {X 0,Y 523.939,Z 204.219,A -85,B 0,C 180,E1 -4877.97,E2 -4877.97} C_VEL
LIN {X 0,Y 523.965,Z 204.214,A -85,B 0,C 180,E1 -4880.411,E2 -4880.411} C_VEL
LIN {X 0,Y 523.908,Z 204.219,A -85,B 0,C 180,E1 -4882.894,E2 -4882.894} C_VEL
LIN {X 0,Y 523.946,Z 204.22,A -85,B 0,C 180,E1 -4885.419,E2 -4885.419} C_VEL
LIN {X 0,Y 523.951,Z 204.215,A -85,B 0,C 180,E1 -4888,E2 -4888} C_VEL
LIN {X 0,Y 523.939,Z 204.217,A -85,B 0,C 180,E1 -4890.856,E2 -4890.856} C_VEL
LIN {X 0,Y 523.955,Z 204.215,A -85,B 0,C 180,E1 -4893.736,E2 -4893.736} C_VEL
LIN {X 0,Y 523.915,Z 204.221,A -85,B 0,C 180,E1 -4896.405,E2 -4896.405} C_VEL
LIN {X 0,Y 523.919,Z 204.225,A -85,B 0,C 180,E1 -4899.085,E2 -4899.085} C_VEL
LIN {X 0,Y 523.95,Z 204.214,A -85,B 0,C 180,E1 -4902.12,E2 -4902.12} C_VEL
LIN {X 0,Y 523.953,Z 204.219,A -85,B 0,C 180,E1 -4905.31,E2 -4905.31} C_VEL
LIN {X 0,Y 523.917,Z 204.226,A -85,B 0,C 180,E1 -4906.91,E2 -4906.91} C_VEL
LIN {X 0,Y 523.251,Z 204.305,A -85,B 0,C 180,E1 -4907.551,E2 -4907.551} C_VEL
LIN {X 0,Y 520.408,Z 204.661,A -85,B 0,C 180,E1 -4908.593,E2 -4908.593} C_VEL
LIN {X 0,Y 518.003,Z 204.957,A -85,B 0,C 180,E1 -4909.432,E2 -4909.432} C_VEL
LIN {X 0,Y 516.966,Z 205.085,A -85,B 0,C 180,E1 -4910.08,E2 -4910.08} C_VEL
LIN {X 0,Y 516.879,Z 205.097,A -85,B 0,C 180,E1 -4910.299,E2 -4910.299} C_VEL
LIN {X 0,Y 516.875,Z 205.099,A -85,B 0,C 180,E1 -4913.344,E2 -4913.344} C_VEL
LIN {X 0,Y 516.914,Z 205.096,A -85,B 0,C 180,E1 -4916.122,E2 -4916.122} C_VEL
LIN {X 0,Y 516.862,Z 205.126,A -85,B 0,C 180,E1 -4918.334,E2 -4918.334} C_VEL
LIN {X 0,Y 517.029,Z 222.118,A -85,B 0,C 180,E1 -4920.67,E2 -4920.67} C_VEL
LIN {X 0,Y 519.141,Z 235.014,A -85,B 0,C 180,E1 -4920.917,E2 -4920.917} C_VEL
LIN {X 0,Y 518.607,Z 330.687,A -85,B 0,C 180,E1 -4922.264,E2 -4922.264} C_VEL
LIN {X 0,Y 518.394,Z 344.134,A -85,B 0,C 180,E1 -4922.608,E2 -4922.608} C_VEL
LIN {X 0,Y 518.204,Z 356.416,A -85,B 0,C 180,E1 -4923.088,E2 -4923.088} C_VEL
LIN {X 0,Y 517.988,Z 367.855,A -85,B 0,C 180,E1 -4923.688,E2 -4923.688} C_VEL
LIN {X 0,Y 517.631,Z 379.454,A -85,B 0,C 180,E1 -4924.465,E2 -4924.465} C_VEL
LIN {X 0,Y 517.367,Z 390.004,A -85,B 0,C 180,E1 -4925.367,E2 -4925.367} C_VEL
LIN {X 0,Y 517.05,Z 399.471,A -85,B 0,C 180,E1 -4926.362,E2 -4926.362} C_VEL
LIN {X 0,Y 516.858,Z 407.61,A -85,B 0,C 180,E1 -4927.411,E2 -4927.411} C_VEL
LIN {X 0,Y 516.596,Z 415.39,A -85,B 0,C 180,E1 -4928.66,E2 -4928.66} C_VEL
LIN {X 0,Y 516.481,Z 421.402,A -85,B 0,C 180,E1 -4929.872,E2 -4929.872} C_VEL
LIN {X 0,Y 516.386,Z 425.601,A -85,B 0,C 180,E1 -4930.936,E2 -4930.936} C_VEL
LIN {X 0,Y 516.307,Z 429.787,A -85,B 0,C 180,E1 -4932.336,E2 -4932.336} C_VEL
LIN {X 0,Y 516.222,Z 431.972,A -85,B 0,C 180,E1 -4933.388,E2 -4933.388} C_VEL
LIN {X 0,Y 516.173,Z 433.179,A -85,B 0,C 180,E1 -4934.199,E2 -4934.199} C_VEL
LIN {X 0,Y 516.206,Z 434.001,A -85,B 0,C 180,E1 -4935.162,E2 -4935.162} C_VEL
LIN {X 0,Y 516.196,Z 434.165,A -85,B 0,C 180,E1 -4936.618,E2 -4936.618} C_VEL
LIN {X 0,Y 516.228,Z 433.645,A -85,B 0,C 180,E1 -4937.42,E2 -4937.42} C_VEL
LIN {X 0,Y 516.287,Z 432.222,A -85,B 0,C 180,E1 -4938.555,E2 -4938.555} C_VEL
LIN {X 0,Y 516.339,Z 428.577,A -85,B 0,C 180,E1 -4940.205,E2 -4940.205} C_VEL
LIN {X 0,Y 516.418,Z 424.736,A -85,B 0,C 180,E1 -4941.391,E2 -4941.391} C_VEL
LIN {X 0,Y 516.524,Z 419.774,A -85,B 0,C 180,E1 -4942.574,E2 -4942.574} C_VEL
LIN {X 0,Y 516.673,Z 413.517,A -85,B 0,C 180,E1 -4943.754,E2 -4943.754} C_VEL
LIN {X 0,Y 516.87,Z 405.743,A -85,B 0,C 180,E1 -4944.93,E2 -4944.93} C_VEL
LIN {X 0,Y 517.086,Z 397.838,A -85,B 0,C 180,E1 -4945.909,E2 -4945.909} C_VEL
LIN {X 0,Y 517.392,Z 388.237,A -85,B 0,C 180,E1 -4946.886,E2 -4946.886} C_VEL
LIN {X 0,Y 517.664,Z 377.493,A -85,B 0,C 180,E1 -4947.764,E2 -4947.764} C_VEL
LIN {X 0,Y 518.015,Z 365.416,A -85,B 0,C 180,E1 -4948.543,E2 -4948.543} C_VEL
LIN {X 0,Y 518.235,Z 353.535,A -85,B 0,C 180,E1 -4949.127,E2 -4949.127} C_VEL
LIN {X 0,Y 518.511,Z 340.494,A -85,B 0,C 180,E1 -4949.588,E2 -4949.588} C_VEL
LIN {X 0,Y 518.652,Z 327.793,A -85,B 0,C 180,E1 -4949.88,E2 -4949.88} C_VEL
LIN {X 0,Y 519.087,Z 233.958,A -85,B 0,C 180,E1 -4951.189,E2 -4951.189} C_VEL
LIN {X 0,Y 517.025,Z 222.023,A -85,B 0,C 180,E1 -4951.437,E2 -4951.437} C_VEL
LIN {X 0,Y 516.838,Z 205.11,A -85,B 0,C 180,E1 -4953.851,E2 -4953.851} C_VEL
LIN {X 0,Y 516.989,Z 205.084,A -85,B 0,C 180,E1 -4956.244,E2 -4956.244} C_VEL
LIN {X 0,Y 516.94,Z 205.095,A -85,B 0,C 180,E1 -4959.39,E2 -4959.39} C_VEL
LIN {X 0,Y 516.959,Z 205.089,A -85,B 0,C 180,E1 -4961.807,E2 -4961.807} C_VEL
LIN {X 0,Y 516.943,Z 205.095,A -85,B 0,C 180,E1 -4965.143,E2 -4965.143} C_VEL
LIN {X 0,Y 516.919,Z 205.093,A -85,B 0,C 180,E1 -4968.223,E2 -4968.223} C_VEL
LIN {X 0,Y 516.911,Z 205.098,A -85,B 0,C 180,E1 -4970.702,E2 -4970.702} C_VEL
LIN {X 0,Y 516.89,Z 205.096,A -85,B 0,C 180,E1 -4974.074,E2 -4974.074} C_VEL
LIN {X 0,Y 516.841,Z 205.108,A -85,B 0,C 180,E1 -4976.663,E2 -4976.663} C_VEL
LIN {X 0,Y 516.893,Z 205.096,A -85,B 0,C 180,E1 -4979.519,E2 -4979.519} C_VEL
LIN {X 0,Y 516.896,Z 205.101,A -85,B 0,C 180,E1 -4982.542,E2 -4982.542} C_VEL
LIN {X 0,Y 516.859,Z 205.101,A -85,B 0,C 180,E1 -4985.328,E2 -4985.328} C_VEL
LIN {X 0,Y 516.864,Z 205.101,A -85,B 0,C 180,E1 -4987.94,E2 -4987.94} C_VEL
LIN {X 0,Y 516.825,Z 205.109,A -85,B 0,C 180,E1 -4990.748,E2 -4990.748} C_VEL
LIN {X 0,Y 516.866,Z 205.102,A -85,B 0,C 180,E1 -4993.906,E2 -4993.906} C_VEL
LIN {X 0,Y 516.865,Z 205.105,A -85,B 0,C 180,E1 -4996.11,E2 -4996.11} C_VEL
LIN {X 0,Y 516.824,Z 205.104,A -85,B 0,C 180,E1 -4999.252,E2 -4999.252} C_VEL
LIN {X 0,Y 516.831,Z 205.108,A -85,B 0,C 180,E1 -5002.065,E2 -5002.065} C_VEL
LIN {X 0,Y 516.855,Z 205.101,A -85,B 0,C 180,E1 -5005.173,E2 -5005.173} C_VEL
LIN {X 0,Y 516.851,Z 205.106,A -85,B 0,C 180,E1 -5007.973,E2 -5007.973} C_VEL
LIN {X 0,Y 516.836,Z 205.103,A -85,B 0,C 180,E1 -5010.69,E2 -5010.69} C_VEL
LIN {X 0,Y 516.833,Z 205.106,A -85,B 0,C 180,E1 -5013.337,E2 -5013.337} C_VEL
LIN {X 0,Y 516.89,Z 205.101,A -85,B 0,C 180,E1 -5015.927,E2 -5015.927} C_VEL
LIN {X 0,Y 516.917,Z 205.098,A -85,B 0,C 180,E1 -5019.298,E2 -5019.298} C_VEL
LIN {X 0,Y 516.977,Z 205.216,A -85,B 0,C 180,E1 -5019.768,E2 -5019.768} C_VEL
LIN {X 0,Y 517.453,Z 210.929,A -85,B 0,C 180,E1 -5020.976,E2 -5020.976} C_VEL
LIN {X 0,Y 517.217,Z 224.285,A -85,B 0,C 180,E1 -5023.711,E2 -5023.711} C_VEL
LIN {X 0,Y 519.077,Z 234.116,A -85,B 0,C 180,E1 -5023.921,E2 -5023.921} C_VEL
LIN {X 0,Y 518.456,Z 331.815,A -85,B 0,C 180,E1 -5025.376,E2 -5025.376} C_VEL
LIN {X 0,Y 518.287,Z 345.382,A -85,B 0,C 180,E1 -5025.747,E2 -5025.747} C_VEL
LIN {X 0,Y 518.114,Z 357.136,A -85,B 0,C 180,E1 -5026.218,E2 -5026.218} C_VEL
LIN {X 0,Y 517.78,Z 369.08,A -85,B 0,C 180,E1 -5026.858,E2 -5026.858} C_VEL
LIN {X 0,Y 517.537,Z 380.442,A -85,B 0,C 180,E1 -5027.642,E2 -5027.642} C_VEL
LIN {X 0,Y 517.279,Z 390.855,A -85,B 0,C 180,E1 -5028.539,E2 -5028.539} C_VEL
LIN {X 0,Y 516.995,Z 400.913,A -85,B 0,C 180,E1 -5029.623,E2 -5029.623} C_VEL
LIN {X 0,Y 516.758,Z 409.747,A -85,B 0,C 180,E1 -5030.804,E2 -5030.804} C_VEL
LIN {X 0,Y 516.584,Z 416.778,A -85,B 0,C 180,E1 -5031.984,E2 -5031.984} C_VEL
LIN {X 0,Y 516.461,Z 422.612,A -85,B 0,C 180,E1 -5033.214,E2 -5033.214} C_VEL
LIN {X 0,Y 516.389,Z 427.424,A -85,B 0,C 180,E1 -5034.533,E2 -5034.533} C_VEL
LIN {X 0,Y 516.289,Z 429.647,A -85,B 0,C 180,E1 -5035.315,E2 -5035.315} C_VEL
LIN {X 0,Y 516.347,Z 431.389,A -85,B 0,C 180,E1 -5036.098,E2 -5036.098} C_VEL
LIN {X 0,Y 516.349,Z 432.73,A -85,B 0,C 180,E1 -5036.879,E2 -5036.879} C_VEL
LIN {X 0,Y 516.265,Z 433.662,A -85,B 0,C 180,E1 -5037.659,E2 -5037.659} C_VEL
LIN {X 0,Y 516.195,Z 434.194,A -85,B 0,C 180,E1 -5038.439,E2 -5038.439} C_VEL
LIN {X 0,Y 516.176,Z 434.307,A -85,B 0,C 180,E1 -5039.22,E2 -5039.22} C_VEL
LIN {X 0,Y 516.184,Z 433.348,A -85,B 0,C 180,E1 -5040.78,E2 -5040.78} C_VEL
LIN {X 0,Y 516.205,Z 432.273,A -85,B 0,C 180,E1 -5041.56,E2 -5041.56} C_VEL
LIN {X 0,Y 516.29,Z 430.749,A -85,B 0,C 180,E1 -5042.34,E2 -5042.34} C_VEL
LIN {X 0,Y 516.434,Z 427.666,A -85,B 0,C 180,E1 -5043.511,E2 -5043.511} C_VEL
LIN {X 0,Y 516.515,Z 423.524,A -85,B 0,C 180,E1 -5044.683,E2 -5044.683} C_VEL
LIN {X 0,Y 516.573,Z 418.204,A -85,B 0,C 180,E1 -5045.856,E2 -5045.856} C_VEL
LIN {X 0,Y 516.711,Z 411.518,A -85,B 0,C 180,E1 -5047.031,E2 -5047.031} C_VEL
LIN {X 0,Y 516.897,Z 403.196,A -85,B 0,C 180,E1 -5048.208,E2 -5048.208} C_VEL
LIN {X 0,Y 517.197,Z 394.593,A -85,B 0,C 180,E1 -5049.187,E2 -5049.187} C_VEL
LIN {X 0,Y 517.433,Z 383.975,A -85,B 0,C 180,E1 -5050.17,E2 -5050.17} C_VEL
LIN {X 0,Y 517.733,Z 373.41,A -85,B 0,C 180,E1 -5050.955,E2 -5050.955} C_VEL
LIN {X 0,Y 517.986,Z 361.626,A -85,B 0,C 180,E1 -5051.643,E2 -5051.643} C_VEL
LIN {X 0,Y 518.242,Z 349.113,A -85,B 0,C 180,E1 -5052.194,E2 -5052.194} C_VEL
LIN {X 0,Y 518.307,Z 336.886,A -85,B 0,C 180,E1 -5052.58,E2 -5052.58} C_VEL
LIN {X 0,Y 518.417,Z 324.218,A -85,B 0,C 180,E1 -5052.826,E2 -5052.826} C_VEL
LIN {X 0,Y 519.068,Z 234.859,A -85,B 0,C 180,E1 -5054.156,E2 -5054.156} C_VEL
LIN {X 0,Y 517.337,Z 225.269,A -85,B 0,C 180,E1 -5054.38,E2 -5054.38} C_VEL
LIN {X 0,Y 517.686,Z 212.927,A -85,B 0,C 180,E1 -5056.97,E2 -5056.97} C_VEL
LIN {X 0,Y 517.467,Z 207.894,A -85,B 0,C 180,E1 -5058.063,E2 -5058.063} C_VEL
LIN {X 0,Y 516.921,Z 205.099,A -85,B 0,C 180,E1 -5058.736,E2 -5058.736} C_VEL
LIN {X 0,Y 516.891,Z 205.098,A -85,B 0,C 180,E1 -5061.537,E2 -5061.537} C_VEL
LIN {X 0,Y 516.89,Z 205.103,A -85,B 0,C 180,E1 -5064.357,E2 -5064.357} C_VEL
LIN {X 0,Y 516.928,Z 205.097,A -85,B 0,C 180,E1 -5066.658,E2 -5066.658} C_VEL
LIN {X 0,Y 516.915,Z 205.094,A -85,B 0,C 180,E1 -5069.523,E2 -5069.523} C_VEL
LIN {X 0,Y 516.901,Z 205.1,A -85,B 0,C 180,E1 -5072.543,E2 -5072.543} C_VEL
LIN {X 0,Y 516.871,Z 205.098,A -85,B 0,C 180,E1 -5075.329,E2 -5075.329} C_VEL
LIN {X 0,Y 516.885,Z 205.101,A -85,B 0,C 180,E1 -5077.943,E2 -5077.943} C_VEL
LIN {X 0,Y 516.888,Z 205.097,A -85,B 0,C 180,E1 -5080.741,E2 -5080.741} C_VEL
LIN {X 0,Y 516.887,Z 205.097,A -85,B 0,C 180,E1 -5082.831,E2 -5082.831} C_VEL
LIN {X 0,Y 516.9,Z 205.094,A -85,B 0,C 180,E1 -5085.007,E2 -5085.007} C_VEL
LIN {X 0,Y 516.913,Z 205.097,A -85,B 0,C 180,E1 -5088.399,E2 -5088.399} C_VEL
LIN {X 0,Y 516.884,Z 205.097,A -85,B 0,C 180,E1 -5091.283,E2 -5091.283} C_VEL
LIN {X 0,Y 516.872,Z 205.103,A -85,B 0,C 180,E1 -5094.219,E2 -5094.219} C_VEL
LIN {X 0,Y 516.9,Z 205.097,A -85,B 0,C 180,E1 -5097.053,E2 -5097.053} C_VEL
LIN {X 0,Y 516.897,Z 205.106,A -85,B 0,C 180,E1 -5099.796,E2 -5099.796} C_VEL
LIN {X 0,Y 516.897,Z 205.1,A -85,B 0,C 180,E1 -5102.465,E2 -5102.465} C_VEL
LIN {X 0,Y 516.96,Z 205.235,A -85,B 0,C 180,E1 -5104.859,E2 -5104.859} C_VEL
LIN {X 0,Y 518.416,Z 213.199,A -85,B 0,C 180,E1 -5106.214,E2 -5106.214} C_VEL
LIN {X 0,Y 518.256,Z 223.842,A -85,B 0,C 180,E1 -5107.894,E2 -5107.894} C_VEL
LIN {X 0,Y 517.717,Z 243.94,A -85,B 0,C 180,E1 -5110.985,E2 -5110.985} C_VEL
LIN {X 0,Y 517.319,Z 261.483,A -85,B 0,C 180,E1 -5113.626,E2 -5113.626} C_VEL
LIN {X 0,Y 517.231,Z 268.255,A -85,B 0,C 180,E1 -5114.639,E2 -5114.639} C_VEL
LIN {X 0,Y 518.954,Z 281.47,A -85,B 0,C 180,E1 -5114.898,E2 -5114.898} C_VEL
LIN {X 0,Y 518.339,Z 378.367,A -85,B 0,C 180,E1 -5116.348,E2 -5116.348} C_VEL
LIN {X 0,Y 518.09,Z 391.926,A -85,B 0,C 180,E1 -5116.716,E2 -5116.716} C_VEL
LIN {X 0,Y 517.849,Z 404.259,A -85,B 0,C 180,E1 -5117.209,E2 -5117.209} C_VEL
LIN {X 0,Y 517.634,Z 415.989,A -85,B 0,C 180,E1 -5117.839,E2 -5117.839} C_VEL
LIN {X 0,Y 517.28,Z 427.669,A -85,B 0,C 180,E1 -5118.637,E2 -5118.637} C_VEL
LIN {X 0,Y 517.069,Z 438.025,A -85,B 0,C 180,E1 -5119.525,E2 -5119.525} C_VEL
LIN {X 0,Y 516.796,Z 448.152,A -85,B 0,C 180,E1 -5120.607,E2 -5120.607} C_VEL
LIN {X 0,Y 516.592,Z 457.076,A -85,B 0,C 180,E1 -5121.787,E2 -5121.787} C_VEL
LIN {X 0,Y 516.438,Z 464.171,A -85,B 0,C 180,E1 -5122.964,E2 -5122.964} C_VEL
LIN {X 0,Y 516.381,Z 469.846,A -85,B 0,C 180,E1 -5124.14,E2 -5124.14} C_VEL
LIN {X 0,Y 516.268,Z 474.298,A -85,B 0,C 180,E1 -5125.314,E2 -5125.314} C_VEL
LIN {X 0,Y 516.37,Z 476.663,A -85,B 0,C 180,E1 -5126.097,E2 -5126.097} C_VEL
LIN {X 0,Y 516.282,Z 478.578,A -85,B 0,C 180,E1 -5126.878,E2 -5126.878} C_VEL
LIN {X 0,Y 516.261,Z 480.011,A -85,B 0,C 180,E1 -5127.659,E2 -5127.659} C_VEL
LIN {X 0,Y 516.167,Z 481.659,A -85,B 0,C 180,E1 -5129.219,E2 -5129.219} C_VEL
LIN {X 0,Y 516.167,Z 481.89,A -85,B 0,C 180,E1 -5129.999,E2 -5129.999} C_VEL
LIN {X 0,Y 516.167,Z 481.676,A -85,B 0,C 180,E1 -5130.779,E2 -5130.779} C_VEL
LIN {X 0,Y 516.261,Z 480.062,A -85,B 0,C 180,E1 -5132.34,E2 -5132.34} C_VEL
LIN {X 0,Y 516.282,Z 478.643,A -85,B 0,C 180,E1 -5133.12,E2 -5133.12} C_VEL
LIN {X 0,Y 516.311,Z 475.667,A -85,B 0,C 180,E1 -5134.293,E2 -5134.293} C_VEL
LIN {X 0,Y 516.367,Z 471.632,A -85,B 0,C 180,E1 -5135.466,E2 -5135.466} C_VEL
LIN {X 0,Y 516.414,Z 466.352,A -85,B 0,C 180,E1 -5136.655,E2 -5136.655} C_VEL
LIN {X 0,Y 516.542,Z 459.85,A -85,B 0,C 180,E1 -5137.819,E2 -5137.819} C_VEL
LIN {X 0,Y 516.754,Z 451.672,A -85,B 0,C 180,E1 -5138.997,E2 -5138.997} C_VEL
LIN {X 0,Y 516.918,Z 443.311,A -85,B 0,C 180,E1 -5139.982,E2 -5139.982} C_VEL
LIN {X 0,Y 517.22,Z 433.075,A -85,B 0,C 180,E1 -5140.965,E2 -5140.965} C_VEL
LIN {X 0,Y 517.511,Z 421.612,A -85,B 0,C 180,E1 -5141.843,E2 -5141.843} C_VEL
LIN {X 0,Y 517.788,Z 410.1,A -85,B 0,C 180,E1 -5142.542,E2 -5142.542} C_VEL
LIN {X 0,Y 518.059,Z 398.486,A -85,B 0,C 180,E1 -5143.083,E2 -5143.083} C_VEL
LIN {X 0,Y 518.293,Z 386.066,A -85,B 0,C 180,E1 -5143.501,E2 -5143.501} C_VEL
LIN {X 0,Y 518.471,Z 372.336,A -85,B 0,C 180,E1 -5143.796,E2 -5143.796} C_VEL
LIN {X 0,Y 518.87,Z 280.051,A -85,B 0,C 180,E1 -5145.138,E2 -5145.138} C_VEL
LIN {X 0,Y 517.27,Z 269.076,A -85,B 0,C 180,E1 -5145.365,E2 -5145.365} C_VEL
LIN {X 0,Y 517.747,Z 249.08,A -85,B 0,C 180,E1 -5148.396,E2 -5148.396} C_VEL
LIN {X 0,Y 518.327,Z 227.591,A -85,B 0,C 180,E1 -5151.683,E2 -5151.683} C_VEL
LIN {X 0,Y 518.698,Z 214.26,A -85,B 0,C 180,E1 -5153.771,E2 -5153.771} C_VEL
LIN {X 0,Y 516.955,Z 205.093,A -85,B 0,C 180,E1 -5155.328,E2 -5155.328} C_VEL
LIN {X 0,Y 516.907,Z 205.098,A -85,B 0,C 180,E1 -5158.415,E2 -5158.415} C_VEL
LIN {X 0,Y 516.886,Z 205.096,A -85,B 0,C 180,E1 -5161.109,E2 -5161.109} C_VEL
LIN {X 0,Y 516.904,Z 205.089,A -85,B 0,C 180,E1 -5163.965,E2 -5163.965} C_VEL
LIN {X 0,Y 516.848,Z 205.1,A -85,B 0,C 180,E1 -5166.747,E2 -5166.747} C_VEL
LIN {X 0,Y 516.854,Z 205.104,A -85,B 0,C 180,E1 -5169.723,E2 -5169.723} C_VEL
LIN {X 0,Y 516.896,Z 205.099,A -85,B 0,C 180,E1 -5171.775,E2 -5171.775} C_VEL
LIN {X 0,Y 516.889,Z 205.095,A -85,B 0,C 180,E1 -5175.006,E2 -5175.006} C_VEL
LIN {X 0,Y 516.881,Z 205.09,A -85,B 0,C 180,E1 -5178.401,E2 -5178.401} C_VEL
LIN {X 0,Y 516.869,Z 205.104,A -85,B 0,C 180,E1 -5181.283,E2 -5181.283} C_VEL
LIN {X 0,Y 516.863,Z 205.091,A -85,B 0,C 180,E1 -5184.219,E2 -5184.219} C_VEL
LIN {X 0,Y 516.872,Z 205.101,A -85,B 0,C 180,E1 -5187.051,E2 -5187.051} C_VEL
LIN {X 0,Y 516.854,Z 205.093,A -85,B 0,C 180,E1 -5189.794,E2 -5189.794} C_VEL
LIN {X 0,Y 516.865,Z 205.094,A -85,B 0,C 180,E1 -5192.464,E2 -5192.464} C_VEL
LIN {X 0,Y 516.834,Z 205.106,A -85,B 0,C 180,E1 -5195.068,E2 -5195.068} C_VEL
LIN {X 0,Y 516.86,Z 205.089,A -85,B 0,C 180,E1 -5197.621,E2 -5197.621} C_VEL
LIN {X 0,Y 516.904,Z 205.09,A -85,B 0,C 180,E1 -5200.129,E2 -5200.129} C_VEL
LIN {X 0,Y 516.862,Z 205.096,A -85,B 0,C 180,E1 -5203.409,E2 -5203.409} C_VEL
LIN {X 0,Y 516.857,Z 205.09,A -85,B 0,C 180,E1 -5205.833,E2 -5205.833} C_VEL
LIN {X 0,Y 516.933,Z 205.092,A -85,B 0,C 180,E1 -5209.028,E2 -5209.028} C_VEL
LIN {X 0,Y 516.932,Z 205.093,A -85,B 0,C 180,E1 -5212.186,E2 -5212.186} C_VEL
LIN {X 0,Y 516.972,Z 205.082,A -85,B 0,C 180,E1 -5214.54,E2 -5214.54} C_VEL
LIN {X 0,Y 517.064,Z 205.072,A -85,B 0,C 180,E1 -5217.663,E2 -5217.663} C_VEL
LIN {X 0,Y 517.081,Z 205.068,A -85,B 0,C 180,E1 -5220.779,E2 -5220.779} C_VEL
LIN {X 0,Y 516.962,Z 205.076,A -85,B 0,C 180,E1 -5223.117,E2 -5223.117} C_VEL
LIN {X 0,Y 516.997,Z 205.086,A -85,B 0,C 180,E1 -5226.244,E2 -5226.244} C_VEL
LIN {X 0,Y 516.933,Z 205.085,A -85,B 0,C 180,E1 -5229.39,E2 -5229.39} C_VEL
LIN {X 0,Y 516.944,Z 205.087,A -85,B 0,C 180,E1 -5231.807,E2 -5231.807} C_VEL
LIN {X 0,Y 516.937,Z 205.088,A -85,B 0,C 180,E1 -5235.147,E2 -5235.147} C_VEL
LIN {X 0,Y 516.908,Z 205.092,A -85,B 0,C 180,E1 -5238.223,E2 -5238.223} C_VEL
LIN {X 0,Y 516.905,Z 205.092,A -85,B 0,C 180,E1 -5240.702,E2 -5240.702} C_VEL
LIN {X 0,Y 516.905,Z 205.092,A -85,B 0,C 180,E1 -5244.073,E2 -5244.073} C_VEL
LIN {X 0,Y 516.916,Z 205.092,A -85,B 0,C 180,E1 -5246.659,E2 -5246.659} C_VEL
LIN {X 0,Y 516.904,Z 205.096,A -85,B 0,C 180,E1 -5249.524,E2 -5249.524} C_VEL
LIN {X 0,Y 516.89,Z 205.095,A -85,B 0,C 180,E1 -5252.544,E2 -5252.544} C_VEL
LIN {X 0,Y 516.875,Z 205.104,A -85,B 0,C 180,E1 -5255.333,E2 -5255.333} C_VEL
LIN {X 0,Y 516.877,Z 205.095,A -85,B 0,C 180,E1 -5257.944,E2 -5257.944} C_VEL
LIN {X 0,Y 516.881,Z 205.101,A -85,B 0,C 180,E1 -5260.743,E2 -5260.743} C_VEL
LIN {X 0,Y 516.88,Z 205.1,A -85,B 0,C 180,E1 -5262.832,E2 -5262.832} C_VEL
LIN {X 0,Y 516.92,Z 205.097,A -85,B 0,C 180,E1 -5265.011,E2 -5265.011} C_VEL
LIN {X 0,Y 516.914,Z 205.094,A -85,B 0,C 180,E1 -5268.399,E2 -5268.399} C_VEL
LIN {X 0,Y 516.879,Z 205.097,A -85,B 0,C 180,E1 -5270.299,E2 -5270.299} C_VEL
LIN {X 0,Y 516.208,Z 205.186,A -85,B 0,C 180,E1 -5270.949,E2 -5270.949} C_VEL
LIN {X 0,Y 513.362,Z 205.54,A -85,B 0,C 180,E1 -5272.005,E2 -5272.005} C_VEL
LIN {X 0,Y 510.952,Z 205.841,A -85,B 0,C 180,E1 -5272.855,E2 -5272.855} C_VEL
LIN {X 0,Y 509.909,Z 205.966,A -85,B 0,C 180,E1 -5273.511,E2 -5273.511} C_VEL
LIN {X 0,Y 509.819,Z 205.977,A -85,B 0,C 180,E1 -5273.734,E2 -5273.734} C_VEL
LIN {X 0,Y 509.872,Z 205.977,A -85,B 0,C 180,E1 -5276.541,E2 -5276.541} C_VEL
LIN {X 0,Y 509.815,Z 206.045,A -85,B 0,C 180,E1 -5278.309,E2 -5278.309} C_VEL
LIN {X 0,Y 509.996,Z 221.967,A -85,B 0,C 180,E1 -5280.442,E2 -5280.442} C_VEL
LIN {X 0,Y 512.305,Z 236.179,A -85,B 0,C 180,E1 -5280.724,E2 -5280.724} C_VEL
LIN {X 0,Y 511.715,Z 331.756,A -85,B 0,C 180,E1 -5282.092,E2 -5282.092} C_VEL
LIN {X 0,Y 511.492,Z 344.566,A -85,B 0,C 180,E1 -5282.429,E2 -5282.429} C_VEL
LIN {X 0,Y 511.301,Z 356.821,A -85,B 0,C 180,E1 -5282.916,E2 -5282.916} C_VEL
LIN {X 0,Y 511.049,Z 369.267,A -85,B 0,C 180,E1 -5283.585,E2 -5283.585} C_VEL
LIN {X 0,Y 510.701,Z 379.83,A -85,B 0,C 180,E1 -5284.312,E2 -5284.312} C_VEL
LIN {X 0,Y 510.399,Z 389.016,A -85,B 0,C 180,E1 -5285.093,E2 -5285.093} C_VEL
LIN {X 0,Y 510.138,Z 397.995,A -85,B 0,C 180,E1 -5286.021,E2 -5286.021} C_VEL
LIN {X 0,Y 509.854,Z 406.429,A -85,B 0,C 180,E1 -5287.083,E2 -5287.083} C_VEL
LIN {X 0,Y 509.603,Z 414.583,A -85,B 0,C 180,E1 -5288.352,E2 -5288.352} C_VEL
LIN {X 0,Y 509.422,Z 421.519,A -85,B 0,C 180,E1 -5289.741,E2 -5289.741} C_VEL
LIN {X 0,Y 509.301,Z 426.659,A -85,B 0,C 180,E1 -5291.079,E2 -5291.079} C_VEL
LIN {X 0,Y 509.231,Z 430.202,A -85,B 0,C 180,E1 -5292.325,E2 -5292.325} C_VEL
LIN {X 0,Y 509.176,Z 431.93,A -85,B 0,C 180,E1 -5293.152,E2 -5293.152} C_VEL
LIN {X 0,Y 509.086,Z 433.225,A -85,B 0,C 180,E1 -5293.973,E2 -5293.973} C_VEL
LIN {X 0,Y 509.121,Z 434.276,A -85,B 0,C 180,E1 -5295.084,E2 -5295.084} C_VEL
LIN {X 0,Y 509.101,Z 434.518,A -85,B 0,C 180,E1 -5296.428,E2 -5296.428} C_VEL
LIN {X 0,Y 509.139,Z 434.13,A -85,B 0,C 180,E1 -5297.241,E2 -5297.241} C_VEL
LIN {X 0,Y 509.191,Z 432.658,A -85,B 0,C 180,E1 -5298.514,E2 -5298.514} C_VEL
LIN {X 0,Y 509.252,Z 429.397,A -85,B 0,C 180,E1 -5300.067,E2 -5300.067} C_VEL
LIN {X 0,Y 509.328,Z 425.725,A -85,B 0,C 180,E1 -5301.271,E2 -5301.271} C_VEL
LIN {X 0,Y 509.449,Z 420.945,A -85,B 0,C 180,E1 -5302.47,E2 -5302.47} C_VEL
LIN {X 0,Y 509.605,Z 414.931,A -85,B 0,C 180,E1 -5303.667,E2 -5303.667} C_VEL
LIN {X 0,Y 509.806,Z 407.442,A -85,B 0,C 180,E1 -5304.86,E2 -5304.86} C_VEL
LIN {X 0,Y 510.082,Z 398.093,A -85,B 0,C 180,E1 -5306.051,E2 -5306.051} C_VEL
LIN {X 0,Y 510.439,Z 388.468,A -85,B 0,C 180,E1 -5307.041,E2 -5307.041} C_VEL
LIN {X 0,Y 510.738,Z 377.699,A -85,B 0,C 180,E1 -5307.931,E2 -5307.931} C_VEL
LIN {X 0,Y 511.101,Z 365.6,A -85,B 0,C 180,E1 -5308.72,E2 -5308.72} C_VEL
LIN {X 0,Y 511.331,Z 353.669,A -85,B 0,C 180,E1 -5309.312,E2 -5309.312} C_VEL
LIN {X 0,Y 511.624,Z 340.56,A -85,B 0,C 180,E1 -5309.78,E2 -5309.78} C_VEL
LIN {X 0,Y 511.77,Z 327.634,A -85,B 0,C 180,E1 -5310.075,E2 -5310.075} C_VEL
LIN {X 0,Y 512.221,Z 234.687,A -85,B 0,C 180,E1 -5311.389,E2 -5311.389} C_VEL
LIN {X 0,Y 510.004,Z 222.011,A -85,B 0,C 180,E1 -5311.654,E2 -5311.654} C_VEL
LIN {X 0,Y 509.802,Z 205.986,A -85,B 0,C 180,E1 -5313.879,E2 -5313.879} C_VEL
LIN {X 0,Y 509.943,Z 205.962,A -85,B 0,C 180,E1 -5316.331,E2 -5316.331} C_VEL
LIN {X 0,Y 509.906,Z 205.967,A -85,B 0,C 180,E1 -5318.721,E2 -5318.721} C_VEL
LIN {X 0,Y 509.911,Z 205.967,A -85,B 0,C 180,E1 -5321.932,E2 -5321.932} C_VEL
LIN {X 0,Y 509.902,Z 205.971,A -85,B 0,C 180,E1 -5325.242,E2 -5325.242} C_VEL
LIN {X 0,Y 509.864,Z 205.973,A -85,B 0,C 180,E1 -5328.484,E2 -5328.484} C_VEL
LIN {X 0,Y 509.852,Z 205.978,A -85,B 0,C 180,E1 -5331.002,E2 -5331.002} C_VEL
LIN {X 0,Y 509.825,Z 205.978,A -85,B 0,C 180,E1 -5333.565,E2 -5333.565} C_VEL
LIN {X 0,Y 509.813,Z 205.98,A -85,B 0,C 180,E1 -5336.355,E2 -5336.355} C_VEL
LIN {X 0,Y 509.843,Z 205.978,A -85,B 0,C 180,E1 -5338.847,E2 -5338.847} C_VEL
LIN {X 0,Y 509.818,Z 205.977,A -85,B 0,C 180,E1 -5341.591,E2 -5341.591} C_VEL
LIN {X 0,Y 509.838,Z 205.98,A -85,B 0,C 180,E1 -5344.415,E2 -5344.415} C_VEL
LIN {X 0,Y 509.796,Z 205.98,A -85,B 0,C 180,E1 -5347.343,E2 -5347.343} C_VEL
LIN {X 0,Y 509.791,Z 205.985,A -85,B 0,C 180,E1 -5350.388,E2 -5350.388} C_VEL
LIN {X 0,Y 509.798,Z 205.98,A -85,B 0,C 180,E1 -5353.575,E2 -5353.575} C_VEL
LIN {X 0,Y 509.796,Z 205.984,A -85,B 0,C 180,E1 -5356.425,E2 -5356.425} C_VEL
LIN {X 0,Y 509.791,Z 205.982,A -85,B 0,C 180,E1 -5359.613,E2 -5359.613} C_VEL
LIN {X 0,Y 509.756,Z 205.987,A -85,B 0,C 180,E1 -5362.653,E2 -5362.653} C_VEL
LIN {X 0,Y 509.833,Z 205.98,A -85,B 0,C 180,E1 -5365.802,E2 -5365.802} C_VEL
LIN {X 0,Y 509.841,Z 205.975,A -85,B 0,C 180,E1 -5368.722,E2 -5368.722} C_VEL
LIN {X 0,Y 509.827,Z 205.981,A -85,B 0,C 180,E1 -5372.05,E2 -5372.05} C_VEL
LIN {X 0,Y 509.794,Z 205.98,A -85,B 0,C 180,E1 -5374.699,E2 -5374.699} C_VEL
LIN {X 0,Y 509.832,Z 205.981,A -85,B 0,C 180,E1 -5377.458,E2 -5377.458} C_VEL
LIN {X 0,Y 509.947,Z 206.135,A -85,B 0,C 180,E1 -5379.646,E2 -5379.646} C_VEL
LIN {X 0,Y 510.454,Z 211.054,A -85,B 0,C 180,E1 -5380.704,E2 -5380.704} C_VEL
LIN {X 0,Y 510.28,Z 223.024,A -85,B 0,C 180,E1 -5383.188,E2 -5383.188} C_VEL
LIN {X 0,Y 510.241,Z 224.527,A -85,B 0,C 180,E1 -5383.496,E2 -5383.496} C_VEL
LIN {X 0,Y 512.262,Z 235.945,A -85,B 0,C 180,E1 -5383.744,E2 -5383.744} C_VEL
LIN {X 0,Y 511.546,Z 331.798,A -85,B 0,C 180,E1 -5385.199,E2 -5385.199} C_VEL
LIN {X 0,Y 511.366,Z 344.678,A -85,B 0,C 180,E1 -5385.55,E2 -5385.55} C_VEL
LIN {X 0,Y 511.17,Z 356.683,A -85,B 0,C 180,E1 -5386.027,E2 -5386.027} C_VEL
LIN {X 0,Y 510.848,Z 368.842,A -85,B 0,C 180,E1 -5386.677,E2 -5386.677} C_VEL
LIN {X 0,Y 510.556,Z 380.317,A -85,B 0,C 180,E1 -5387.472,E2 -5387.472} C_VEL
LIN {X 0,Y 510.298,Z 390.812,A -85,B 0,C 180,E1 -5388.38,E2 -5388.38} C_VEL
LIN {X 0,Y 510.021,Z 399.302,A -85,B 0,C 180,E1 -5389.279,E2 -5389.279} C_VEL
LIN {X 0,Y 509.756,Z 408.477,A -85,B 0,C 180,E1 -5390.477,E2 -5390.477} C_VEL
LIN {X 0,Y 509.563,Z 415.854,A -85,B 0,C 180,E1 -5391.673,E2 -5391.673} C_VEL
LIN {X 0,Y 509.421,Z 421.757,A -85,B 0,C 180,E1 -5392.867,E2 -5392.867} C_VEL
LIN {X 0,Y 509.386,Z 426.392,A -85,B 0,C 180,E1 -5394.06,E2 -5394.06} C_VEL
LIN {X 0,Y 509.203,Z 429.914,A -85,B 0,C 180,E1 -5395.25,E2 -5395.25} C_VEL
LIN {X 0,Y 509.275,Z 431.677,A -85,B 0,C 180,E1 -5396.043,E2 -5396.043} C_VEL
LIN {X 0,Y 509.26,Z 433.02,A -85,B 0,C 180,E1 -5396.835,E2 -5396.835} C_VEL
LIN {X 0,Y 509.197,Z 433.97,A -85,B 0,C 180,E1 -5397.627,E2 -5397.627} C_VEL
LIN {X 0,Y 509.116,Z 434.524,A -85,B 0,C 180,E1 -5398.418,E2 -5398.418} C_VEL
LIN {X 0,Y 509.087,Z 434.357,A -85,B 0,C 180,E1 -5400,E2 -5400} C_VEL
LIN {X 0,Y 509.096,Z 433.692,A -85,B 0,C 180,E1 -5400.791,E2 -5400.791} C_VEL
LIN {X 0,Y 509.125,Z 432.622,A -85,B 0,C 180,E1 -5401.582,E2 -5401.582} C_VEL
LIN {X 0,Y 509.221,Z 431.094,A -85,B 0,C 180,E1 -5402.373,E2 -5402.373} C_VEL
LIN {X 0,Y 509.371,Z 428.011,A -85,B 0,C 180,E1 -5403.56,E2 -5403.56} C_VEL
LIN {X 0,Y 509.443,Z 423.865,A -85,B 0,C 180,E1 -5404.748,E2 -5404.748} C_VEL
LIN {X 0,Y 509.533,Z 418.534,A -85,B 0,C 180,E1 -5405.938,E2 -5405.938} C_VEL
LIN {X 0,Y 509.679,Z 411.832,A -85,B 0,C 180,E1 -5407.129,E2 -5407.129} C_VEL
LIN {X 0,Y 509.877,Z 403.488,A -85,B 0,C 180,E1 -5408.321,E2 -5408.321} C_VEL
LIN {X 0,Y 510.206,Z 394.858,A -85,B 0,C 180,E1 -5409.314,E2 -5409.314} C_VEL
LIN {X 0,Y 510.45,Z 384.209,A -85,B 0,C 180,E1 -5410.311,E2 -5410.311} C_VEL
LIN {X 0,Y 510.783,Z 373.613,A -85,B 0,C 180,E1 -5411.106,E2 -5411.106} C_VEL
LIN {X 0,Y 511.031,Z 361.775,A -85,B 0,C 180,E1 -5411.804,E2 -5411.804} C_VEL
LIN {X 0,Y 511.308,Z 348.905,A -85,B 0,C 180,E1 -5412.374,E2 -5412.374} C_VEL
LIN {X 0,Y 511.391,Z 336.915,A -85,B 0,C 180,E1 -5412.753,E2 -5412.753} C_VEL
LIN {X 0,Y 511.556,Z 322.348,A -85,B 0,C 180,E1 -5413.026,E2 -5413.026} C_VEL
LIN {X 0,Y 512.229,Z 236.012,A -85,B 0,C 180,E1 -5414.349,E2 -5414.349} C_VEL
LIN {X 0,Y 510.367,Z 225.771,A -85,B 0,C 180,E1 -5414.58,E2 -5414.58} C_VEL
LIN {X 0,Y 510.774,Z 213.487,A -85,B 0,C 180,E1 -5417.207,E2 -5417.207} C_VEL
LIN {X 0,Y 510.468,Z 209.001,A -85,B 0,C 180,E1 -5418.198,E2 -5418.198} C_VEL
LIN {X 0,Y 509.889,Z 205.974,A -85,B 0,C 180,E1 -5418.899,E2 -5418.899} C_VEL
LIN {X 0,Y 509.856,Z 205.977,A -85,B 0,C 180,E1 -5421.001,E2 -5421.001} C_VEL
LIN {X 0,Y 509.827,Z 205.977,A -85,B 0,C 180,E1 -5423.564,E2 -5423.564} C_VEL
LIN {X 0,Y 509.915,Z 205.972,A -85,B 0,C 180,E1 -5426.378,E2 -5426.378} C_VEL
LIN {X 0,Y 509.88,Z 205.972,A -85,B 0,C 180,E1 -5428.844,E2 -5428.844} C_VEL
LIN {X 0,Y 509.824,Z 205.977,A -85,B 0,C 180,E1 -5431.59,E2 -5431.59} C_VEL
LIN {X 0,Y 509.852,Z 205.978,A -85,B 0,C 180,E1 -5434.413,E2 -5434.413} C_VEL
LIN {X 0,Y 509.822,Z 205.977,A -85,B 0,C 180,E1 -5437.34,E2 -5437.34} C_VEL
LIN {X 0,Y 509.843,Z 205.978,A -85,B 0,C 180,E1 -5440.382,E2 -5440.382} C_VEL
LIN {X 0,Y 509.827,Z 205.976,A -85,B 0,C 180,E1 -5443.062,E2 -5443.062} C_VEL
LIN {X 0,Y 509.827,Z 205.98,A -85,B 0,C 180,E1 -5445.793,E2 -5445.793} C_VEL
LIN {X 0,Y 509.856,Z 205.974,A -85,B 0,C 180,E1 -5448.574,E2 -5448.574} C_VEL
LIN {X 0,Y 509.854,Z 205.977,A -85,B 0,C 180,E1 -5451.786,E2 -5451.786} C_VEL
LIN {X 0,Y 509.832,Z 205.977,A -85,B 0,C 180,E1 -5454.621,E2 -5454.621} C_VEL
LIN {X 0,Y 509.866,Z 205.976,A -85,B 0,C 180,E1 -5457.48,E2 -5457.48} C_VEL
LIN {X 0,Y 509.863,Z 205.98,A -85,B 0,C 180,E1 -5460.273,E2 -5460.273} C_VEL
LIN {X 0,Y 509.88,Z 205.975,A -85,B 0,C 180,E1 -5463.629,E2 -5463.629} C_VEL
LIN {X 0,Y 509.865,Z 206.027,A -85,B 0,C 180,E1 -5464.621,E2 -5464.621} C_VEL
LIN {X 0,Y 511.478,Z 214.394,A -85,B 0,C 180,E1 -5466.086,E2 -5466.086} C_VEL
LIN {X 0,Y 511.4,Z 222.329,A -85,B 0,C 180,E1 -5467.368,E2 -5467.368} C_VEL
LIN {X 0,Y 510.865,Z 238.313,A -85,B 0,C 180,E1 -5469.883,E2 -5469.883} C_VEL
LIN {X 0,Y 510.466,Z 255.721,A -85,B 0,C 180,E1 -5472.575,E2 -5472.575} C_VEL
LIN {X 0,Y 510.214,Z 267.773,A -85,B 0,C 180,E1 -5474.407,E2 -5474.407} C_VEL
LIN {X 0,Y 512.105,Z 283.109,A -85,B 0,C 180,E1 -5474.724,E2 -5474.724} C_VEL
LIN {X 0,Y 511.413,Z 378.075,A -85,B 0,C 180,E1 -5476.185,E2 -5476.185} C_VEL
LIN {X 0,Y 511.149,Z 391.592,A -85,B 0,C 180,E1 -5476.558,E2 -5476.558} C_VEL
LIN {X 0,Y 510.865,Z 404.41,A -85,B 0,C 180,E1 -5477.081,E2 -5477.081} C_VEL
LIN {X 0,Y 510.623,Z 416.463,A -85,B 0,C 180,E1 -5477.746,E2 -5477.746} C_VEL
LIN {X 0,Y 510.227,Z 428.303,A -85,B 0,C 180,E1 -5478.579,E2 -5478.579} C_VEL
LIN {X 0,Y 510.013,Z 438.432,A -85,B 0,C 180,E1 -5479.479,E2 -5479.479} C_VEL
LIN {X 0,Y 509.717,Z 447.622,A -85,B 0,C 180,E1 -5480.475,E2 -5480.475} C_VEL
LIN {X 0,Y 509.517,Z 456.595,A -85,B 0,C 180,E1 -5481.672,E2 -5481.672} C_VEL
LIN {X 0,Y 509.391,Z 463.737,A -85,B 0,C 180,E1 -5482.866,E2 -5482.866} C_VEL
LIN {X 0,Y 509.28,Z 469.44,A -85,B 0,C 180,E1 -5484.058,E2 -5484.058} C_VEL
LIN {X 0,Y 509.186,Z 473.918,A -85,B 0,C 180,E1 -5485.249,E2 -5485.249} C_VEL
LIN {X 0,Y 509.275,Z 476.298,A -85,B 0,C 180,E1 -5486.043,E2 -5486.043} C_VEL
LIN {X 0,Y 509.201,Z 478.225,A -85,B 0,C 180,E1 -5486.834,E2 -5486.834} C_VEL
LIN {X 0,Y 509.19,Z 479.669,A -85,B 0,C 180,E1 -5487.626,E2 -5487.626} C_VEL
LIN {X 0,Y 509.08,Z 481.331,A -85,B 0,C 180,E1 -5489.208,E2 -5489.208} C_VEL
LIN {X 0,Y 509.078,Z 481.565,A -85,B 0,C 180,E1 -5489.999,E2 -5489.999} C_VEL
LIN {X 0,Y 509.08,Z 481.351,A -85,B 0,C 180,E1 -5490.79,E2 -5490.79} C_VEL
LIN {X 0,Y 509.19,Z 479.735,A -85,B 0,C 180,E1 -5492.372,E2 -5492.372} C_VEL
LIN {X 0,Y 509.201,Z 478.309,A -85,B 0,C 180,E1 -5493.164,E2 -5493.164} C_VEL
LIN {X 0,Y 509.204,Z 475.322,A -85,B 0,C 180,E1 -5494.353,E2 -5494.353} C_VEL
LIN {X 0,Y 509.279,Z 471.273,A -85,B 0,C 180,E1 -5495.542,E2 -5495.542} C_VEL
LIN {X 0,Y 509.366,Z 465.124,A -85,B 0,C 180,E1 -5496.913,E2 -5496.913} C_VEL
LIN {X 0,Y 509.489,Z 458.194,A -85,B 0,C 180,E1 -5498.127,E2 -5498.127} C_VEL
LIN {X 0,Y 509.706,Z 449.709,A -85,B 0,C 180,E1 -5499.323,E2 -5499.323} C_VEL
LIN {X 0,Y 509.929,Z 440.957,A -85,B 0,C 180,E1 -5500.32,E2 -5500.32} C_VEL
LIN {X 0,Y 510.306,Z 430.187,A -85,B 0,C 180,E1 -5501.317,E2 -5501.317} C_VEL
LIN {X 0,Y 510.494,Z 419.574,A -85,B 0,C 180,E1 -5502.111,E2 -5502.111} C_VEL
LIN {X 0,Y 510.854,Z 407.512,A -85,B 0,C 180,E1 -5502.816,E2 -5502.816} C_VEL
LIN {X 0,Y 511.144,Z 395.114,A -85,B 0,C 180,E1 -5503.365,E2 -5503.365} C_VEL
LIN {X 0,Y 511.456,Z 382.424,A -85,B 0,C 180,E1 -5503.761,E2 -5503.761} C_VEL
LIN {X 0,Y 511.6,Z 367.649,A -85,B 0,C 180,E1 -5504.036,E2 -5504.036} C_VEL
LIN {X 0,Y 512.007,Z 280.704,A -85,B 0,C 180,E1 -5505.331,E2 -5505.331} C_VEL
LIN {X 0,Y 510.255,Z 268.854,A -85,B 0,C 180,E1 -5505.573,E2 -5505.573} C_VEL
LIN {X 0,Y 510.771,Z 248.799,A -85,B 0,C 180,E1 -5508.656,E2 -5508.656} C_VEL
LIN {X 0,Y 511.402,Z 228.738,A -85,B 0,C 180,E1 -5511.779,E2 -5511.779} C_VEL
LIN {X 0,Y 511.719,Z 215.354,A -85,B 0,C 180,E1 -5513.9,E2 -5513.9} C_VEL
LIN {X 0,Y 509.916,Z 205.97,A -85,B 0,C 180,E1 -5515.511,E2 -5515.511} C_VEL
LIN {X 0,Y 509.869,Z 205.971,A -85,B 0,C 180,E1 -5518.844,E2 -5518.844} C_VEL
LIN {X 0,Y 509.817,Z 205.98,A -85,B 0,C 180,E1 -5521.589,E2 -5521.589} C_VEL
LIN {X 0,Y 509.843,Z 205.969,A -85,B 0,C 180,E1 -5524.413,E2 -5524.413} C_VEL
LIN {X 0,Y 509.803,Z 205.98,A -85,B 0,C 180,E1 -5527.341,E2 -5527.341} C_VEL
LIN {X 0,Y 509.812,Z 205.977,A -85,B 0,C 180,E1 -5530.383,E2 -5530.383} C_VEL
LIN {X 0,Y 509.798,Z 205.978,A -85,B 0,C 180,E1 -5533.059,E2 -5533.059} C_VEL
LIN {X 0,Y 509.816,Z 205.981,A -85,B 0,C 180,E1 -5535.793,E2 -5535.793} C_VEL
LIN {X 0,Y 509.825,Z 205.969,A -85,B 0,C 180,E1 -5538.571,E2 -5538.571} C_VEL
LIN {X 0,Y 509.842,Z 205.974,A -85,B 0,C 180,E1 -5541.786,E2 -5541.786} C_VEL
LIN {X 0,Y 509.821,Z 205.968,A -85,B 0,C 180,E1 -5544.621,E2 -5544.621} C_VEL
LIN {X 0,Y 509.849,Z 205.975,A -85,B 0,C 180,E1 -5547.48,E2 -5547.48} C_VEL
LIN {X 0,Y 509.844,Z 205.965,A -85,B 0,C 180,E1 -5550.275,E2 -5550.275} C_VEL
LIN {X 0,Y 509.814,Z 205.978,A -85,B 0,C 180,E1 -5552.94,E2 -5552.94} C_VEL
LIN {X 0,Y 509.824,Z 205.972,A -85,B 0,C 180,E1 -5555.572,E2 -5555.572} C_VEL
LIN {X 0,Y 509.806,Z 205.966,A -85,B 0,C 180,E1 -5558.148,E2 -5558.148} C_VEL
LIN {X 0,Y 509.835,Z 205.976,A -85,B 0,C 180,E1 -5560.681,E2 -5560.681} C_VEL
LIN {X 0,Y 509.835,Z 205.974,A -85,B 0,C 180,E1 -5563.173,E2 -5563.173} C_VEL
LIN {X 0,Y 509.831,Z 205.964,A -85,B 0,C 180,E1 -5565.633,E2 -5565.633} C_VEL
LIN {X 0,Y 509.897,Z 205.97,A -85,B 0,C 180,E1 -5568.874,E2 -5568.874} C_VEL
LIN {X 0,Y 509.897,Z 205.968,A -85,B 0,C 180,E1 -5572.078,E2 -5572.078} C_VEL
LIN {X 0,Y 509.87,Z 205.961,A -85,B 0,C 180,E1 -5575.256,E2 -5575.256} C_VEL
LIN {X 0,Y 510.035,Z 205.947,A -85,B 0,C 180,E1 -5577.631,E2 -5577.631} C_VEL
LIN {X 0,Y 510.051,Z 205.943,A -85,B 0,C 180,E1 -5580.79,E2 -5580.79} C_VEL
LIN {X 0,Y 509.905,Z 205.955,A -85,B 0,C 180,E1 -5583.161,E2 -5583.161} C_VEL
LIN {X 0,Y 509.948,Z 205.963,A -85,B 0,C 180,E1 -5586.33,E2 -5586.33} C_VEL
LIN {X 0,Y 509.901,Z 205.961,A -85,B 0,C 180,E1 -5588.721,E2 -5588.721} C_VEL
LIN {X 0,Y 509.896,Z 205.967,A -85,B 0,C 180,E1 -5591.932,E2 -5591.932} C_VEL
LIN {X 0,Y 509.886,Z 205.967,A -85,B 0,C 180,E1 -5595.242,E2 -5595.242} C_VEL
LIN {X 0,Y 509.853,Z 205.968,A -85,B 0,C 180,E1 -5598.484,E2 -5598.484} C_VEL
LIN {X 0,Y 509.843,Z 205.973,A -85,B 0,C 180,E1 -5601.002,E2 -5601.002} C_VEL
LIN {X 0,Y 509.863,Z 205.966,A -85,B 0,C 180,E1 -5604.427,E2 -5604.427} C_VEL
LIN {X 0,Y 509.875,Z 205.972,A -85,B 0,C 180,E1 -5607.057,E2 -5607.057} C_VEL
LIN {X 0,Y 509.851,Z 205.974,A -85,B 0,C 180,E1 -5609.752,E2 -5609.752} C_VEL
LIN {X 0,Y 509.868,Z 205.972,A -85,B 0,C 180,E1 -5612.775,E2 -5612.775} C_VEL
LIN {X 0,Y 509.835,Z 205.979,A -85,B 0,C 180,E1 -5615.582,E2 -5615.582} C_VEL
LIN {X 0,Y 509.846,Z 205.97,A -85,B 0,C 180,E1 -5618.339,E2 -5618.339} C_VEL
LIN {X 0,Y 509.853,Z 205.973,A -85,B 0,C 180,E1 -5621.426,E2 -5621.426} C_VEL
LIN {X 0,Y 509.854,Z 205.976,A -85,B 0,C 180,E1 -5624.669,E2 -5624.669} C_VEL
LIN {X 0,Y 509.856,Z 205.971,A -85,B 0,C 180,E1 -5628.104,E2 -5628.104} C_VEL
LIN {X 0,Y 509.844,Z 205.978,A -85,B 0,C 180,E1 -5630.649,E2 -5630.649} C_VEL
LIN {X 0,Y 509.819,Z 205.977,A -85,B 0,C 180,E1 -5633.734,E2 -5633.734} C_VEL
LIN {X 0,Y 509.141,Z 206.066,A -85,B 0,C 180,E1 -5634.394,E2 -5634.394} C_VEL
LIN {X 0,Y 506.297,Z 206.421,A -85,B 0,C 180,E1 -5635.466,E2 -5635.466} C_VEL
LIN {X 0,Y 503.917,Z 206.719,A -85,B 0,C 180,E1 -5636.329,E2 -5636.329} C_VEL
LIN {X 0,Y 502.916,Z 206.843,A -85,B 0,C 180,E1 -5636.996,E2 -5636.996} C_VEL
LIN {X 0,Y 502.845,Z 206.85,A -85,B 0,C 180,E1 -5637.221,E2 -5637.221} C_VEL
LIN {X 0,Y 502.785,Z 206.898,A -85,B 0,C 180,E1 -5638.251,E2 -5638.251} C_VEL
LIN {X 0,Y 502.982,Z 221.987,A -85,B 0,C 180,E1 -5640.215,E2 -5640.215} C_VEL
LIN {X 0,Y 505.419,Z 235.702,A -85,B 0,C 180,E1 -5640.497,E2 -5640.497} C_VEL
LIN {X 0,Y 504.837,Z 331.783,A -85,B 0,C 180,E1 -5641.892,E2 -5641.892} C_VEL
LIN {X 0,Y 504.598,Z 345.049,A -85,B 0,C 180,E1 -5642.245,E2 -5642.245} C_VEL
LIN {X 0,Y 504.362,Z 358.099,A -85,B 0,C 180,E1 -5642.779,E2 -5642.779} C_VEL
LIN {X 0,Y 504.128,Z 369.294,A -85,B 0,C 180,E1 -5643.394,E2 -5643.394} C_VEL
LIN {X 0,Y 503.747,Z 380.209,A -85,B 0,C 180,E1 -5644.153,E2 -5644.153} C_VEL
LIN {X 0,Y 503.414,Z 390.372,A -85,B 0,C 180,E1 -5645.043,E2 -5645.043} C_VEL
LIN {X 0,Y 503.074,Z 400.182,A -85,B 0,C 180,E1 -5646.102,E2 -5646.102} C_VEL
LIN {X 0,Y 502.801,Z 409.093,A -85,B 0,C 180,E1 -5647.3,E2 -5647.3} C_VEL
LIN {X 0,Y 502.506,Z 417.221,A -85,B 0,C 180,E1 -5648.678,E2 -5648.678} C_VEL
LIN {X 0,Y 502.335,Z 423.27,A -85,B 0,C 180,E1 -5649.993,E2 -5649.993} C_VEL
LIN {X 0,Y 502.219,Z 427.646,A -85,B 0,C 180,E1 -5651.226,E2 -5651.226} C_VEL
LIN {X 0,Y 502.158,Z 430.133,A -85,B 0,C 180,E1 -5652.122,E2 -5652.122} C_VEL
LIN {X 0,Y 502.107,Z 431.883,A -85,B 0,C 180,E1 -5652.907,E2 -5652.907} C_VEL
LIN {X 0,Y 502.029,Z 433.264,A -85,B 0,C 180,E1 -5653.742,E2 -5653.742} C_VEL
LIN {X 0,Y 502.026,Z 434.554,A -85,B 0,C 180,E1 -5655.007,E2 -5655.007} C_VEL
LIN {X 0,Y 502.021,Z 434.871,A -85,B 0,C 180,E1 -5656.233,E2 -5656.233} C_VEL
LIN {X 0,Y 502.03,Z 434.561,A -85,B 0,C 180,E1 -5657.058,E2 -5657.058} C_VEL
LIN {X 0,Y 502.11,Z 433.088,A -85,B 0,C 180,E1 -5658.463,E2 -5658.463} C_VEL
LIN {X 0,Y 502.147,Z 431.146,A -85,B 0,C 180,E1 -5659.518,E2 -5659.518} C_VEL
LIN {X 0,Y 502.193,Z 427.989,A -85,B 0,C 180,E1 -5660.74,E2 -5660.74} C_VEL
LIN {X 0,Y 502.325,Z 423.766,A -85,B 0,C 180,E1 -5661.958,E2 -5661.958} C_VEL
LIN {X 0,Y 502.479,Z 418.024,A -85,B 0,C 180,E1 -5663.247,E2 -5663.247} C_VEL
LIN {X 0,Y 502.728,Z 410.369,A -85,B 0,C 180,E1 -5664.586,E2 -5664.586} C_VEL
LIN {X 0,Y 502.985,Z 401.708,A -85,B 0,C 180,E1 -5665.794,E2 -5665.794} C_VEL
LIN {X 0,Y 503.32,Z 391.799,A -85,B 0,C 180,E1 -5666.899,E2 -5666.899} C_VEL
LIN {X 0,Y 503.639,Z 381.784,A -85,B 0,C 180,E1 -5667.802,E2 -5667.802} C_VEL
LIN {X 0,Y 504.073,Z 370.703,A -85,B 0,C 180,E1 -5668.603,E2 -5668.603} C_VEL
LIN {X 0,Y 504.36,Z 359.161,A -85,B 0,C 180,E1 -5669.252,E2 -5669.252} C_VEL
LIN {X 0,Y 504.611,Z 347.432,A -85,B 0,C 180,E1 -5669.752,E2 -5669.752} C_VEL
LIN {X 0,Y 504.821,Z 334.919,A -85,B 0,C 180,E1 -5670.126,E2 -5670.126} C_VEL
LIN {X 0,Y 504.979,Z 318.792,A -85,B 0,C 180,E1 -5670.4,E2 -5670.4} C_VEL
LIN {X 0,Y 505.435,Z 235.967,A -85,B 0,C 180,E1 -5671.582,E2 -5671.582} C_VEL
LIN {X 0,Y 502.976,Z 221.97,A -85,B 0,C 180,E1 -5671.878,E2 -5671.878} C_VEL
LIN {X 0,Y 502.785,Z 206.86,A -85,B 0,C 180,E1 -5673.933,E2 -5673.933} C_VEL
LIN {X 0,Y 502.898,Z 206.839,A -85,B 0,C 180,E1 -5676.42,E2 -5676.42} C_VEL
LIN {X 0,Y 502.866,Z 206.845,A -85,B 0,C 180,E1 -5678.844,E2 -5678.844} C_VEL
LIN {X 0,Y 502.852,Z 206.845,A -85,B 0,C 180,E1 -5682.102,E2 -5682.102} C_VEL
LIN {X 0,Y 502.856,Z 206.848,A -85,B 0,C 180,E1 -5685.4,E2 -5685.4} C_VEL
LIN {X 0,Y 502.829,Z 206.852,A -85,B 0,C 180,E1 -5688.753,E2 -5688.753} C_VEL
LIN {X 0,Y 502.787,Z 206.857,A -85,B 0,C 180,E1 -5691.312,E2 -5691.312} C_VEL
LIN {X 0,Y 502.772,Z 206.855,A -85,B 0,C 180,E1 -5693.916,E2 -5693.916} C_VEL
LIN {X 0,Y 502.788,Z 206.858,A -85,B 0,C 180,E1 -5696.571,E2 -5696.571} C_VEL
LIN {X 0,Y 502.816,Z 206.85,A -85,B 0,C 180,E1 -5699.934,E2 -5699.934} C_VEL
LIN {X 0,Y 502.808,Z 206.854,A -85,B 0,C 180,E1 -5703.034,E2 -5703.034} C_VEL
LIN {X 0,Y 502.766,Z 206.857,A -85,B 0,C 180,E1 -5705.953,E2 -5705.953} C_VEL
LIN {X 0,Y 502.776,Z 206.857,A -85,B 0,C 180,E1 -5708.979,E2 -5708.979} C_VEL
LIN {X 0,Y 502.751,Z 206.863,A -85,B 0,C 180,E1 -5712.192,E2 -5712.192} C_VEL
LIN {X 0,Y 502.784,Z 206.854,A -85,B 0,C 180,E1 -5715.471,E2 -5715.471} C_VEL
LIN {X 0,Y 502.755,Z 206.858,A -85,B 0,C 180,E1 -5718.927,E2 -5718.927} C_VEL
LIN {X 0,Y 502.744,Z 206.863,A -85,B 0,C 180,E1 -5722.041,E2 -5722.041} C_VEL
LIN {X 0,Y 502.755,Z 206.857,A -85,B 0,C 180,E1 -5725.03,E2 -5725.03} C_VEL
LIN {X 0,Y 502.766,Z 206.86,A -85,B 0,C 180,E1 -5727.914,E2 -5727.914} C_VEL
LIN {X 0,Y 502.761,Z 206.857,A -85,B 0,C 180,E1 -5730.708,E2 -5730.708} C_VEL
LIN {X 0,Y 502.776,Z 206.859,A -85,B 0,C 180,E1 -5733.461,E2 -5733.461} C_VEL
LIN {X 0,Y 502.772,Z 206.859,A -85,B 0,C 180,E1 -5736.085,E2 -5736.085} C_VEL
LIN {X 0,Y 502.788,Z 206.854,A -85,B 0,C 180,E1 -5738.689,E2 -5738.689} C_VEL
LIN {X 0,Y 502.88,Z 206.945,A -85,B 0,C 180,E1 -5739.497,E2 -5739.497} C_VEL
LIN {X 0,Y 503.476,Z 213.187,A -85,B 0,C 180,E1 -5740.85,E2 -5740.85} C_VEL
LIN {X 0,Y 503.305,Z 225.08,A -85,B 0,C 180,E1 -5743.293,E2 -5743.293} C_VEL
LIN {X 0,Y 505.405,Z 236.473,A -85,B 0,C 180,E1 -5743.541,E2 -5743.541} C_VEL
LIN {X 0,Y 504.64,Z 331.782,A -85,B 0,C 180,E1 -5745.018,E2 -5745.018} C_VEL
LIN {X 0,Y 504.454,Z 344.731,A -85,B 0,C 180,E1 -5745.373,E2 -5745.373} C_VEL
LIN {X 0,Y 504.223,Z 357.351,A -85,B 0,C 180,E1 -5745.882,E2 -5745.882} C_VEL
LIN {X 0,Y 503.916,Z 368.603,A -85,B 0,C 180,E1 -5746.49,E2 -5746.49} C_VEL
LIN {X 0,Y 503.584,Z 380.266,A -85,B 0,C 180,E1 -5747.302,E2 -5747.302} C_VEL
LIN {X 0,Y 503.308,Z 390.756,A -85,B 0,C 180,E1 -5748.216,E2 -5748.216} C_VEL
LIN {X 0,Y 503.035,Z 399.32,A -85,B 0,C 180,E1 -5749.128,E2 -5749.128} C_VEL
LIN {X 0,Y 502.789,Z 407.198,A -85,B 0,C 180,E1 -5750.14,E2 -5750.14} C_VEL
LIN {X 0,Y 502.554,Z 414.867,A -85,B 0,C 180,E1 -5751.353,E2 -5751.353} C_VEL
LIN {X 0,Y 502.374,Z 421.942,A -85,B 0,C 180,E1 -5752.767,E2 -5752.767} C_VEL
LIN {X 0,Y 502.32,Z 426.617,A -85,B 0,C 180,E1 -5753.976,E2 -5753.976} C_VEL
LIN {X 0,Y 502.121,Z 430.171,A -85,B 0,C 180,E1 -5755.182,E2 -5755.182} C_VEL
LIN {X 0,Y 502.204,Z 431.956,A -85,B 0,C 180,E1 -5755.987,E2 -5755.987} C_VEL
LIN {X 0,Y 502.175,Z 433.312,A -85,B 0,C 180,E1 -5756.791,E2 -5756.791} C_VEL
LIN {X 0,Y 502.129,Z 434.275,A -85,B 0,C 180,E1 -5757.593,E2 -5757.593} C_VEL
LIN {X 0,Y 502.04,Z 434.843,A -85,B 0,C 180,E1 -5758.395,E2 -5758.395} C_VEL
LIN {X 0,Y 502.004,Z 434.966,A -85,B 0,C 180,E1 -5759.198,E2 -5759.198} C_VEL
LIN {X 0,Y 502.012,Z 434.033,A -85,B 0,C 180,E1 -5760.802,E2 -5760.802} C_VEL
LIN {X 0,Y 502.049,Z 432.967,A -85,B 0,C 180,E1 -5761.604,E2 -5761.604} C_VEL
LIN {X 0,Y 502.155,Z 431.441,A -85,B 0,C 180,E1 -5762.406,E2 -5762.406} C_VEL
LIN {X 0,Y 502.311,Z 428.356,A -85,B 0,C 180,E1 -5763.61,E2 -5763.61} C_VEL
LIN {X 0,Y 502.374,Z 424.205,A -85,B 0,C 180,E1 -5764.815,E2 -5764.815} C_VEL
LIN {X 0,Y 502.495,Z 418.861,A -85,B 0,C 180,E1 -5766.021,E2 -5766.021} C_VEL
LIN {X 0,Y 502.635,Z 412.15,A -85,B 0,C 180,E1 -5767.229,E2 -5767.229} C_VEL
LIN {X 0,Y 502.867,Z 403.79,A -85,B 0,C 180,E1 -5768.438,E2 -5768.438} C_VEL
LIN {X 0,Y 503.203,Z 395.141,A -85,B 0,C 180,E1 -5769.445,E2 -5769.445} C_VEL
LIN {X 0,Y 503.472,Z 384.474,A -85,B 0,C 180,E1 -5770.455,E2 -5770.455} C_VEL
LIN {X 0,Y 503.832,Z 373.852,A -85,B 0,C 180,E1 -5771.261,E2 -5771.261} C_VEL
LIN {X 0,Y 504.101,Z 361.965,A -85,B 0,C 180,E1 -5771.969,E2 -5771.969} C_VEL
LIN {X 0,Y 504.392,Z 348.675,A -85,B 0,C 180,E1 -5772.562,E2 -5772.562} C_VEL
LIN {X 0,Y 504.476,Z 337.041,A -85,B 0,C 180,E1 -5772.931,E2 -5772.931} C_VEL
LIN {X 0,Y 504.647,Z 322.45,A -85,B 0,C 180,E1 -5773.208,E2 -5773.208} C_VEL
LIN {X 0,Y 505.43,Z 236.39,A -85,B 0,C 180,E1 -5774.565,E2 -5774.565} C_VEL
LIN {X 0,Y 503.425,Z 226.221,A -85,B 0,C 180,E1 -5774.812,E2 -5774.812} C_VEL
LIN {X 0,Y 503.851,Z 214.049,A -85,B 0,C 180,E1 -5777.451,E2 -5777.451} C_VEL
LIN {X 0,Y 503.153,Z 208.463,A -85,B 0,C 180,E1 -5778.739,E2 -5778.739} C_VEL
LIN {X 0,Y 502.829,Z 206.853,A -85,B 0,C 180,E1 -5779.175,E2 -5779.175} C_VEL
LIN {X 0,Y 502.785,Z 206.859,A -85,B 0,C 180,E1 -5782.173,E2 -5782.173} C_VEL
LIN {X 0,Y 502.801,Z 206.856,A -85,B 0,C 180,E1 -5784.792,E2 -5784.792} C_VEL
LIN {X 0,Y 502.836,Z 206.848,A -85,B 0,C 180,E1 -5787.467,E2 -5787.467} C_VEL
LIN {X 0,Y 502.813,Z 206.855,A -85,B 0,C 180,E1 -5790.211,E2 -5790.211} C_VEL
LIN {X 0,Y 502.837,Z 206.847,A -85,B 0,C 180,E1 -5793.031,E2 -5793.031} C_VEL
LIN {X 0,Y 502.778,Z 206.859,A -85,B 0,C 180,E1 -5795.951,E2 -5795.951} C_VEL
LIN {X 0,Y 502.806,Z 206.85,A -85,B 0,C 180,E1 -5798.976,E2 -5798.976} C_VEL
LIN {X 0,Y 502.8,Z 206.857,A -85,B 0,C 180,E1 -5802.139,E2 -5802.139} C_VEL
LIN {X 0,Y 502.79,Z 206.853,A -85,B 0,C 180,E1 -5805.47,E2 -5805.47} C_VEL
LIN {X 0,Y 502.799,Z 206.857,A -85,B 0,C 180,E1 -5807.86,E2 -5807.86} C_VEL
LIN {X 0,Y 502.805,Z 206.85,A -85,B 0,C 180,E1 -5811.023,E2 -5811.023} C_VEL
LIN {X 0,Y 502.776,Z 206.859,A -85,B 0,C 180,E1 -5814.169,E2 -5814.169} C_VEL
LIN {X 0,Y 502.837,Z 206.849,A -85,B 0,C 180,E1 -5816.993,E2 -5816.993} C_VEL
LIN {X 0,Y 502.82,Z 206.86,A -85,B 0,C 180,E1 -5820.064,E2 -5820.064} C_VEL
LIN {X 0,Y 502.848,Z 206.851,A -85,B 0,C 180,E1 -5823.443,E2 -5823.443} C_VEL
LIN {X 0,Y 502.852,Z 206.861,A -85,B 0,C 180,E1 -5824.384,E2 -5824.384} C_VEL
LIN {X 0,Y 504.556,Z 215.634,A -85,B 0,C 180,E1 -5825.956,E2 -5825.956} C_VEL
LIN {X 0,Y 504.492,Z 223.507,A -85,B 0,C 180,E1 -5827.257,E2 -5827.257} C_VEL
LIN {X 0,Y 503.848,Z 240.718,A -85,B 0,C 180,E1 -5830.016,E2 -5830.016} C_VEL
LIN {X 0,Y 503.383,Z 259.451,A -85,B 0,C 180,E1 -5832.95,E2 -5832.95} C_VEL
LIN {X 0,Y 503.199,Z 267.639,A -85,B 0,C 180,E1 -5834.196,E2 -5834.196} C_VEL
LIN {X 0,Y 505.241,Z 282.854,A -85,B 0,C 180,E1 -5834.512,E2 -5834.512} C_VEL
LIN {X 0,Y 504.493,Z 377.896,A -85,B 0,C 180,E1 -5836.017,E2 -5836.017} C_VEL
LIN {X 0,Y 504.204,Z 391.312,A -85,B 0,C 180,E1 -5836.395,E2 -5836.395} C_VEL
LIN {X 0,Y 503.932,Z 403.586,A -85,B 0,C 180,E1 -5836.901,E2 -5836.901} C_VEL
LIN {X 0,Y 503.632,Z 415.978,A -85,B 0,C 180,E1 -5837.589,E2 -5837.589} C_VEL
LIN {X 0,Y 503.219,Z 427.648,A -85,B 0,C 180,E1 -5838.418,E2 -5838.418} C_VEL
LIN {X 0,Y 502.988,Z 437.855,A -85,B 0,C 180,E1 -5839.33,E2 -5839.33} C_VEL
LIN {X 0,Y 502.644,Z 447.092,A -85,B 0,C 180,E1 -5840.34,E2 -5840.34} C_VEL
LIN {X 0,Y 502.463,Z 456.114,A -85,B 0,C 180,E1 -5841.554,E2 -5841.554} C_VEL
LIN {X 0,Y 502.307,Z 463.3,A -85,B 0,C 180,E1 -5842.765,E2 -5842.765} C_VEL
LIN {X 0,Y 502.185,Z 469.037,A -85,B 0,C 180,E1 -5843.974,E2 -5843.974} C_VEL
LIN {X 0,Y 502.109,Z 473.543,A -85,B 0,C 180,E1 -5845.182,E2 -5845.182} C_VEL
LIN {X 0,Y 502.165,Z 475.933,A -85,B 0,C 180,E1 -5845.986,E2 -5845.986} C_VEL
LIN {X 0,Y 502.123,Z 477.873,A -85,B 0,C 180,E1 -5846.79,E2 -5846.79} C_VEL
LIN {X 0,Y 502.121,Z 479.328,A -85,B 0,C 180,E1 -5847.593,E2 -5847.593} C_VEL
LIN {X 0,Y 501.997,Z 481.003,A -85,B 0,C 180,E1 -5849.197,E2 -5849.197} C_VEL
LIN {X 0,Y 501.992,Z 481.239,A -85,B 0,C 180,E1 -5849.999,E2 -5849.999} C_VEL
LIN {X 0,Y 501.996,Z 481.027,A -85,B 0,C 180,E1 -5850.801,E2 -5850.801} C_VEL
LIN {X 0,Y 502.121,Z 479.408,A -85,B 0,C 180,E1 -5852.406,E2 -5852.406} C_VEL
LIN {X 0,Y 502.122,Z 477.976,A -85,B 0,C 180,E1 -5853.209,E2 -5853.209} C_VEL
LIN {X 0,Y 502.102,Z 474.977,A -85,B 0,C 180,E1 -5854.414,E2 -5854.414} C_VEL
LIN {X 0,Y 502.192,Z 470.913,A -85,B 0,C 180,E1 -5855.621,E2 -5855.621} C_VEL
LIN {X 0,Y 502.29,Z 464.739,A -85,B 0,C 180,E1 -5857.011,E2 -5857.011} C_VEL
LIN {X 0,Y 502.426,Z 457.786,A -85,B 0,C 180,E1 -5858.242,E2 -5858.242} C_VEL
LIN {X 0,Y 502.655,Z 449.264,A -85,B 0,C 180,E1 -5859.455,E2 -5859.455} C_VEL
LIN {X 0,Y 502.924,Z 440.478,A -85,B 0,C 180,E1 -5860.466,E2 -5860.466} C_VEL
LIN {X 0,Y 503.285,Z 429.664,A -85,B 0,C 180,E1 -5861.477,E2 -5861.477} C_VEL
LIN {X 0,Y 503.522,Z 418.702,A -85,B 0,C 180,E1 -5862.301,E2 -5862.301} C_VEL
LIN {X 0,Y 503.878,Z 406.844,A -85,B 0,C 180,E1 -5862.997,E2 -5862.997} C_VEL
LIN {X 0,Y 504.202,Z 394.348,A -85,B 0,C 180,E1 -5863.552,E2 -5863.552} C_VEL
LIN {X 0,Y 504.528,Z 381.381,A -85,B 0,C 180,E1 -5863.954,E2 -5863.954} C_VEL
LIN {X 0,Y 504.701,Z 364.547,A -85,B 0,C 180,E1 -5864.258,E2 -5864.258} C_VEL
LIN {X 0,Y 505.143,Z 281.639,A -85,B 0,C 180,E1 -5865.526,E2 -5865.526} C_VEL
LIN {X 0,Y 503.252,Z 268.438,A -85,B 0,C 180,E1 -5865.818,E2 -5865.818} C_VEL
LIN {X 0,Y 503.815,Z 248.518,A -85,B 0,C 180,E1 -5868.924,E2 -5868.924} C_VEL
LIN {X 0,Y 504.454,Z 229.816,A -85,B 0,C 180,E1 -5871.88,E2 -5871.88} C_VEL
LIN {X 0,Y 504.872,Z 217.788,A -85,B 0,C 180,E1 -5873.808,E2 -5873.808} C_VEL
LIN {X 0,Y 502.867,Z 206.85,A -85,B 0,C 180,E1 -5875.701,E2 -5875.701} C_VEL
LIN {X 0,Y 502.834,Z 206.852,A -85,B 0,C 180,E1 -5878.372,E2 -5878.372} C_VEL
LIN {X 0,Y 502.79,Z 206.854,A -85,B 0,C 180,E1 -5881.498,E2 -5881.498} C_VEL
LIN {X 0,Y 502.799,Z 206.844,A -85,B 0,C 180,E1 -5883.993,E2 -5883.993} C_VEL
LIN {X 0,Y 502.76,Z 206.857,A -85,B 0,C 180,E1 -5887.175,E2 -5887.175} C_VEL
LIN {X 0,Y 502.768,Z 206.858,A -85,B 0,C 180,E1 -5890.016,E2 -5890.016} C_VEL
LIN {X 0,Y 502.798,Z 206.85,A -85,B 0,C 180,E1 -5892.198,E2 -5892.198} C_VEL
LIN {X 0,Y 502.779,Z 206.859,A -85,B 0,C 180,E1 -5895.469,E2 -5895.469} C_VEL
LIN {X 0,Y 502.788,Z 206.849,A -85,B 0,C 180,E1 -5897.86,E2 -5897.86} C_VEL
LIN {X 0,Y 502.786,Z 206.855,A -85,B 0,C 180,E1 -5901.022,E2 -5901.022} C_VEL
LIN {X 0,Y 502.767,Z 206.846,A -85,B 0,C 180,E1 -5904.168,E2 -5904.168} C_VEL
LIN {X 0,Y 502.822,Z 206.85,A -85,B 0,C 180,E1 -5906.993,E2 -5906.993} C_VEL
LIN {X 0,Y 502.8,Z 206.842,A -85,B 0,C 180,E1 -5910.066,E2 -5910.066} C_VEL
LIN {X 0,Y 502.774,Z 206.854,A -85,B 0,C 180,E1 -5913.429,E2 -5913.429} C_VEL
LIN {X 0,Y 502.755,Z 206.851,A -85,B 0,C 180,E1 -5916.084,E2 -5916.084} C_VEL
LIN {X 0,Y 502.764,Z 206.848,A -85,B 0,C 180,E1 -5918.688,E2 -5918.688} C_VEL
LIN {X 0,Y 502.796,Z 206.852,A -85,B 0,C 180,E1 -5921.247,E2 -5921.247} C_VEL
LIN {X 0,Y 502.825,Z 206.846,A -85,B 0,C 180,E1 -5924.665,E2 -5924.665} C_VEL
LIN {X 0,Y 502.867,Z 206.838,A -85,B 0,C 180,E1 -5928.039,E2 -5928.039} C_VEL
LIN {X 0,Y 502.848,Z 206.844,A -85,B 0,C 180,E1 -5931.156,E2 -5931.156} C_VEL
LIN {X 0,Y 502.839,Z 206.838,A -85,B 0,C 180,E1 -5933.58,E2 -5933.58} C_VEL
LIN {X 0,Y 502.858,Z 206.843,A -85,B 0,C 180,E1 -5936.795,E2 -5936.795} C_VEL
LIN {X 0,Y 502.89,Z 206.845,A -85,B 0,C 180,E1 -5938.399,E2 -5938.399} C_VEL
LIN {X 0,Y 503.001,Z 206.821,A -85,B 0,C 180,E1 -5940.801,E2 -5940.801} C_VEL
LIN {X 0,Y 503.005,Z 206.818,A -85,B 0,C 180,E1 -5942.403,E2 -5942.403} C_VEL
LIN {X 0,Y 502.921,Z 206.833,A -85,B 0,C 180,E1 -5945.614,E2 -5945.614} C_VEL
LIN {X 0,Y 502.892,Z 206.842,A -85,B 0,C 180,E1 -5948.034,E2 -5948.034} C_VEL
LIN {X 0,Y 502.868,Z 206.834,A -85,B 0,C 180,E1 -5951.284,E2 -5951.284} C_VEL
LIN {X 0,Y 502.836,Z 206.844,A -85,B 0,C 180,E1 -5954.571,E2 -5954.571} C_VEL
LIN {X 0,Y 502.814,Z 206.848,A -85,B 0,C 180,E1 -5957.909,E2 -5957.909} C_VEL
LIN {X 0,Y 502.822,Z 206.847,A -85,B 0,C 180,E1 -5960.537,E2 -5960.537} C_VEL
LIN {X 0,Y 502.787,Z 206.85,A -85,B 0,C 180,E1 -5963.041,E2 -5963.041} C_VEL
LIN {X 0,Y 502.833,Z 206.852,A -85,B 0,C 180,E1 -5965.676,E2 -5965.676} C_VEL
LIN {X 0,Y 502.83,Z 206.843,A -85,B 0,C 180,E1 -5968.374,E2 -5968.374} C_VEL
LIN {X 0,Y 502.787,Z 206.859,A -85,B 0,C 180,E1 -5971.5,E2 -5971.5} C_VEL
LIN {X 0,Y 502.799,Z 206.847,A -85,B 0,C 180,E1 -5974.445,E2 -5974.445} C_VEL
LIN {X 0,Y 502.776,Z 206.86,A -85,B 0,C 180,E1 -5977.179,E2 -5977.179} C_VEL
LIN {X 0,Y 502.784,Z 206.854,A -85,B 0,C 180,E1 -5980.016,E2 -5980.016} C_VEL
LIN {X 0,Y 502.799,Z 206.848,A -85,B 0,C 180,E1 -5982.2,E2 -5982.2} C_VEL
LIN {X 0,Y 502.798,Z 206.853,A -85,B 0,C 180,E1 -5985.469,E2 -5985.469} C_VEL
LIN {X 0,Y 502.818,Z 206.854,A -85,B 0,C 180,E1 -5988.935,E2 -5988.935} C_VEL
LIN {X 0,Y 502.791,Z 206.852,A -85,B 0,C 180,E1 -5992.047,E2 -5992.047} C_VEL
LIN {X 0,Y 502.799,Z 206.856,A -85,B 0,C 180,E1 -5995.035,E2 -5995.035} C_VEL
LIN {X 0,Y 502.845,Z 206.85,A -85,B 0,C 180,E1 -5997.221,E2 -5997.221} C_VEL
LIN {X 0,Y 502.362,Z 207.213,A -85,B 0,C 180,E1 -5997.593,E2 -5997.593} C_VEL
LIN {X 0,Y 500.608,Z 208.649,A -85,B 0,C 180,E1 -5998.067,E2 -5998.067} C_VEL
LIN {X 0,Y 498.118,Z 211.228,A -85,B 0,C 180,E1 -5998.552,E2 -5998.552} C_VEL
LIN {X 0,Y 496.23,Z 214.54,A -85,B 0,C 180,E1 -5999.021,E2 -5999.021} C_VEL
LIN {X 0,Y 495.948,Z 216.376,A -85,B 0,C 180,E1 -5999.258,E2 -5999.258} C_VEL
LIN {X 0,Y 496.065,Z 222.291,A -85,B 0,C 180,E1 -5999.98,E2 -5999.98} C_VEL
LIN {X 0,Y 498.649,Z 237.341,A -85,B 0,C 180,E1 -6000.294,E2 -6000.294} C_VEL
LIN {X 0,Y 498.008,Z 331.265,A -85,B 0,C 180,E1 -6001.673,E2 -6001.673} C_VEL
LIN {X 0,Y 497.774,Z 344.855,A -85,B 0,C 180,E1 -6002.031,E2 -6002.031} C_VEL
LIN {X 0,Y 497.529,Z 357.03,A -85,B 0,C 180,E1 -6002.522,E2 -6002.522} C_VEL
LIN {X 0,Y 497.219,Z 369.78,A -85,B 0,C 180,E1 -6003.223,E2 -6003.223} C_VEL
LIN {X 0,Y 496.82,Z 380.633,A -85,B 0,C 180,E1 -6003.991,E2 -6003.991} C_VEL
LIN {X 0,Y 496.457,Z 390.543,A -85,B 0,C 180,E1 -6004.87,E2 -6004.87} C_VEL
LIN {X 0,Y 496.076,Z 400.554,A -85,B 0,C 180,E1 -6005.965,E2 -6005.965} C_VEL
LIN {X 0,Y 495.791,Z 409.143,A -85,B 0,C 180,E1 -6007.132,E2 -6007.132} C_VEL
LIN {X 0,Y 495.485,Z 416.421,A -85,B 0,C 180,E1 -6008.36,E2 -6008.36} C_VEL
LIN {X 0,Y 495.278,Z 423.086,A -85,B 0,C 180,E1 -6009.779,E2 -6009.779} C_VEL
LIN {X 0,Y 495.151,Z 427.326,A -85,B 0,C 180,E1 -6010.947,E2 -6010.947} C_VEL
LIN {X 0,Y 495.115,Z 430.28,A -85,B 0,C 180,E1 -6011.999,E2 -6011.999} C_VEL
LIN {X 0,Y 494.973,Z 433.3,A -85,B 0,C 180,E1 -6013.503,E2 -6013.503} C_VEL
LIN {X 0,Y 494.943,Z 434.829,A -85,B 0,C 180,E1 -6014.924,E2 -6014.924} C_VEL
LIN {X 0,Y 494.926,Z 435.215,A -85,B 0,C 180,E1 -6016.032,E2 -6016.032} C_VEL
LIN {X 0,Y 494.946,Z 434.991,A -85,B 0,C 180,E1 -6016.869,E2 -6016.869} C_VEL
LIN {X 0,Y 495.023,Z 433.347,A -85,B 0,C 180,E1 -6018.536,E2 -6018.536} C_VEL
LIN {X 0,Y 495.048,Z 431.886,A -85,B 0,C 180,E1 -6019.366,E2 -6019.366} C_VEL
LIN {X 0,Y 495.11,Z 428.89,A -85,B 0,C 180,E1 -6020.606,E2 -6020.606} C_VEL
LIN {X 0,Y 495.257,Z 424.838,A -85,B 0,C 180,E1 -6021.843,E2 -6021.843} C_VEL
LIN {X 0,Y 495.409,Z 418.851,A -85,B 0,C 180,E1 -6023.24,E2 -6023.24} C_VEL
LIN {X 0,Y 495.668,Z 411.929,A -85,B 0,C 180,E1 -6024.509,E2 -6024.509} C_VEL
LIN {X 0,Y 495.931,Z 403.52,A -85,B 0,C 180,E1 -6025.734,E2 -6025.734} C_VEL
LIN {X 0,Y 496.257,Z 394.935,A -85,B 0,C 180,E1 -6026.753,E2 -6026.753} C_VEL
LIN {X 0,Y 496.604,Z 384.428,A -85,B 0,C 180,E1 -6027.77,E2 -6027.77} C_VEL
LIN {X 0,Y 497.067,Z 373.838,A -85,B 0,C 180,E1 -6028.583,E2 -6028.583} C_VEL
LIN {X 0,Y 497.387,Z 362.2,A -85,B 0,C 180,E1 -6029.292,E2 -6029.292} C_VEL
LIN {X 0,Y 497.678,Z 350.165,A -85,B 0,C 180,E1 -6029.849,E2 -6029.849} C_VEL
LIN {X 0,Y 497.92,Z 336.727,A -85,B 0,C 180,E1 -6030.279,E2 -6030.279} C_VEL
LIN {X 0,Y 498.1,Z 323.486,A -85,B 0,C 180,E1 -6030.531,E2 -6030.531} C_VEL
LIN {X 0,Y 498.547,Z 236.358,A -85,B 0,C 180,E1 -6031.793,E2 -6031.793} C_VEL
LIN {X 0,Y 495.967,Z 221.928,A -85,B 0,C 180,E1 -6032.107,E2 -6032.107} C_VEL
LIN {X 0,Y 495.743,Z 207.737,A -85,B 0,C 180,E1 -6033.964,E2 -6033.964} C_VEL
LIN {X 0,Y 495.854,Z 207.717,A -85,B 0,C 180,E1 -6036.512,E2 -6036.512} C_VEL
LIN {X 0,Y 495.836,Z 207.723,A -85,B 0,C 180,E1 -6038.971,E2 -6038.971} C_VEL
LIN {X 0,Y 495.835,Z 207.72,A -85,B 0,C 180,E1 -6042.035,E2 -6042.035} C_VEL
LIN {X 0,Y 495.831,Z 207.723,A -85,B 0,C 180,E1 -6045.452,E2 -6045.452} C_VEL
LIN {X 0,Y 495.785,Z 207.73,A -85,B 0,C 180,E1 -6049.029,E2 -6049.029} C_VEL
LIN {X 0,Y 495.747,Z 207.732,A -85,B 0,C 180,E1 -6051.63,E2 -6051.63} C_VEL
LIN {X 0,Y 495.718,Z 207.735,A -85,B 0,C 180,E1 -6054.278,E2 -6054.278} C_VEL
LIN {X 0,Y 495.736,Z 207.735,A -85,B 0,C 180,E1 -6056.98,E2 -6056.98} C_VEL
LIN {X 0,Y 495.764,Z 207.73,A -85,B 0,C 180,E1 -6060.146,E2 -6060.146} C_VEL
LIN {X 0,Y 495.757,Z 207.731,A -85,B 0,C 180,E1 -6063.237,E2 -6063.237} C_VEL
LIN {X 0,Y 495.71,Z 207.737,A -85,B 0,C 180,E1 -6066.086,E2 -6066.086} C_VEL
LIN {X 0,Y 495.737,Z 207.735,A -85,B 0,C 180,E1 -6068.764,E2 -6068.764} C_VEL
LIN {X 0,Y 495.707,Z 207.737,A -85,B 0,C 180,E1 -6071.787,E2 -6071.787} C_VEL
LIN {X 0,Y 495.737,Z 207.732,A -85,B 0,C 180,E1 -6075.142,E2 -6075.142} C_VEL
LIN {X 0,Y 495.705,Z 207.739,A -85,B 0,C 180,E1 -6078.213,E2 -6078.213} C_VEL
LIN {X 0,Y 495.71,Z 207.736,A -85,B 0,C 180,E1 -6081.404,E2 -6081.404} C_VEL
LIN {X 0,Y 495.716,Z 207.738,A -85,B 0,C 180,E1 -6084.459,E2 -6084.459} C_VEL
LIN {X 0,Y 495.731,Z 207.734,A -85,B 0,C 180,E1 -6087.403,E2 -6087.403} C_VEL
LIN {X 0,Y 495.719,Z 207.738,A -85,B 0,C 180,E1 -6090.25,E2 -6090.25} C_VEL
LIN {X 0,Y 495.726,Z 207.735,A -85,B 0,C 180,E1 -6093.275,E2 -6093.275} C_VEL
LIN {X 0,Y 495.717,Z 207.738,A -85,B 0,C 180,E1 -6095.723,E2 -6095.723} C_VEL
LIN {X 0,Y 495.748,Z 207.732,A -85,B 0,C 180,E1 -6098.371,E2 -6098.371} C_VEL
LIN {X 0,Y 495.819,Z 207.907,A -85,B 0,C 180,E1 -6099.378,E2 -6099.378} C_VEL
LIN {X 0,Y 496.511,Z 213.304,A -85,B 0,C 180,E1 -6100.571,E2 -6100.571} C_VEL
LIN {X 0,Y 496.298,Z 225.207,A -85,B 0,C 180,E1 -6103.071,E2 -6103.071} C_VEL
LIN {X 0,Y 498.578,Z 237.002,A -85,B 0,C 180,E1 -6103.336,E2 -6103.336} C_VEL
LIN {X 0,Y 497.73,Z 332.765,A -85,B 0,C 180,E1 -6104.857,E2 -6104.857} C_VEL
LIN {X 0,Y 497.526,Z 345.468,A -85,B 0,C 180,E1 -6105.217,E2 -6105.217} C_VEL
LIN {X 0,Y 497.286,Z 357.959,A -85,B 0,C 180,E1 -6105.733,E2 -6105.733} C_VEL
LIN {X 0,Y 496.921,Z 369.918,A -85,B 0,C 180,E1 -6106.401,E2 -6106.401} C_VEL
LIN {X 0,Y 496.575,Z 381.792,A -85,B 0,C 180,E1 -6107.255,E2 -6107.255} C_VEL
LIN {X 0,Y 496.296,Z 391.905,A -85,B 0,C 180,E1 -6108.166,E2 -6108.166} C_VEL
LIN {X 0,Y 495.96,Z 401.02,A -85,B 0,C 180,E1 -6109.178,E2 -6109.178} C_VEL
LIN {X 0,Y 495.662,Z 410.029,A -85,B 0,C 180,E1 -6110.409,E2 -6110.409} C_VEL
LIN {X 0,Y 495.436,Z 417.256,A -85,B 0,C 180,E1 -6111.639,E2 -6111.639} C_VEL
LIN {X 0,Y 495.321,Z 422.126,A -85,B 0,C 180,E1 -6112.663,E2 -6112.663} C_VEL
LIN {X 0,Y 495.224,Z 426.15,A -85,B 0,C 180,E1 -6113.695,E2 -6113.695} C_VEL
LIN {X 0,Y 495.045,Z 430.426,A -85,B 0,C 180,E1 -6115.113,E2 -6115.113} C_VEL
LIN {X 0,Y 495.135,Z 432.235,A -85,B 0,C 180,E1 -6115.93,E2 -6115.93} C_VEL
LIN {X 0,Y 495.095,Z 433.607,A -85,B 0,C 180,E1 -6116.745,E2 -6116.745} C_VEL
LIN {X 0,Y 495.064,Z 434.58,A -85,B 0,C 180,E1 -6117.559,E2 -6117.559} C_VEL
LIN {X 0,Y 494.967,Z 435.161,A -85,B 0,C 180,E1 -6118.373,E2 -6118.373} C_VEL
LIN {X 0,Y 494.924,Z 435.297,A -85,B 0,C 180,E1 -6119.186,E2 -6119.186} C_VEL
LIN {X 0,Y 494.931,Z 434.375,A -85,B 0,C 180,E1 -6120.813,E2 -6120.813} C_VEL
LIN {X 0,Y 494.976,Z 433.314,A -85,B 0,C 180,E1 -6121.627,E2 -6121.627} C_VEL
LIN {X 0,Y 495.092,Z 431.79,A -85,B 0,C 180,E1 -6122.441,E2 -6122.441} C_VEL
LIN {X 0,Y 495.237,Z 428.708,A -85,B 0,C 180,E1 -6123.661,E2 -6123.661} C_VEL
LIN {X 0,Y 495.309,Z 424.555,A -85,B 0,C 180,E1 -6124.884,E2 -6124.884} C_VEL
LIN {X 0,Y 495.458,Z 419.206,A -85,B 0,C 180,E1 -6126.107,E2 -6126.107} C_VEL
LIN {X 0,Y 495.604,Z 412.483,A -85,B 0,C 180,E1 -6127.332,E2 -6127.332} C_VEL
LIN {X 0,Y 495.866,Z 404.107,A -85,B 0,C 180,E1 -6128.558,E2 -6128.558} C_VEL
LIN {X 0,Y 496.2,Z 395.453,A -85,B 0,C 180,E1 -6129.58,E2 -6129.58} C_VEL
LIN {X 0,Y 496.5,Z 384.786,A -85,B 0,C 180,E1 -6130.604,E2 -6130.604} C_VEL
LIN {X 0,Y 496.882,Z 374.163,A -85,B 0,C 180,E1 -6131.421,E2 -6131.421} C_VEL
LIN {X 0,Y 497.168,Z 362.278,A -85,B 0,C 180,E1 -6132.138,E2 -6132.138} C_VEL
LIN {X 0,Y 497.467,Z 349.887,A -85,B 0,C 180,E1 -6132.703,E2 -6132.703} C_VEL
LIN {X 0,Y 497.577,Z 337.352,A -85,B 0,C 180,E1 -6133.113,E2 -6133.113} C_VEL
LIN {X 0,Y 497.736,Z 322.892,A -85,B 0,C 180,E1 -6133.394,E2 -6133.394} C_VEL
LIN {X 0,Y 498.634,Z 237.163,A -85,B 0,C 180,E1 -6134.788,E2 -6134.788} C_VEL
LIN {X 0,Y 496.505,Z 226.561,A -85,B 0,C 180,E1 -6135.076,E2 -6135.076} C_VEL
LIN {X 0,Y 496.903,Z 216.584,A -85,B 0,C 180,E1 -6137.278,E2 -6137.278} C_VEL
LIN {X 0,Y 496.493,Z 211.347,A -85,B 0,C 180,E1 -6138.484,E2 -6138.484} C_VEL
LIN {X 0,Y 495.805,Z 207.729,A -85,B 0,C 180,E1 -6139.404,E2 -6139.404} C_VEL
LIN {X 0,Y 495.754,Z 207.735,A -85,B 0,C 180,E1 -6142.505,E2 -6142.505} C_VEL
LIN {X 0,Y 495.785,Z 207.731,A -85,B 0,C 180,E1 -6146.068,E2 -6146.068} C_VEL
LIN {X 0,Y 495.776,Z 207.73,A -85,B 0,C 180,E1 -6148.814,E2 -6148.814} C_VEL
LIN {X 0,Y 495.76,Z 207.73,A -85,B 0,C 180,E1 -6151.725,E2 -6151.725} C_VEL
LIN {X 0,Y 495.774,Z 207.729,A -85,B 0,C 180,E1 -6154.693,E2 -6154.693} C_VEL
LIN {X 0,Y 495.734,Z 207.733,A -85,B 0,C 180,E1 -6157.561,E2 -6157.561} C_VEL
LIN {X 0,Y 495.771,Z 207.728,A -85,B 0,C 180,E1 -6160.699,E2 -6160.699} C_VEL
LIN {X 0,Y 495.733,Z 207.737,A -85,B 0,C 180,E1 -6164.001,E2 -6164.001} C_VEL
LIN {X 0,Y 495.721,Z 207.733,A -85,B 0,C 180,E1 -6167.115,E2 -6167.115} C_VEL
LIN {X 0,Y 495.763,Z 207.733,A -85,B 0,C 180,E1 -6169.953,E2 -6169.953} C_VEL
LIN {X 0,Y 495.723,Z 207.735,A -85,B 0,C 180,E1 -6172.554,E2 -6172.554} C_VEL
LIN {X 0,Y 495.782,Z 207.729,A -85,B 0,C 180,E1 -6175.456,E2 -6175.456} C_VEL
LIN {X 0,Y 495.76,Z 207.736,A -85,B 0,C 180,E1 -6178.363,E2 -6178.363} C_VEL
LIN {X 0,Y 495.759,Z 207.738,A -85,B 0,C 180,E1 -6181.514,E2 -6181.514} C_VEL
LIN {X 0,Y 495.823,Z 207.911,A -85,B 0,C 180,E1 -6184.159,E2 -6184.159} C_VEL
LIN {X 0,Y 497.606,Z 216.917,A -85,B 0,C 180,E1 -6185.82,E2 -6185.82} C_VEL
LIN {X 0,Y 497.686,Z 222.132,A -85,B 0,C 180,E1 -6186.708,E2 -6186.708} C_VEL
LIN {X 0,Y 497.049,Z 237.914,A -85,B 0,C 180,E1 -6189.298,E2 -6189.298} C_VEL
LIN {X 0,Y 496.504,Z 256.501,A -85,B 0,C 180,E1 -6192.281,E2 -6192.281} C_VEL
LIN {X 0,Y 496.165,Z 267.047,A -85,B 0,C 180,E1 -6193.942,E2 -6193.942} C_VEL
LIN {X 0,Y 498.403,Z 284.611,A -85,B 0,C 180,E1 -6194.322,E2 -6194.322} C_VEL
LIN {X 0,Y 497.557,Z 376.809,A -85,B 0,C 180,E1 -6195.818,E2 -6195.818} C_VEL
LIN {X 0,Y 497.291,Z 390.396,A -85,B 0,C 180,E1 -6196.202,E2 -6196.202} C_VEL
LIN {X 0,Y 496.956,Z 402.809,A -85,B 0,C 180,E1 -6196.713,E2 -6196.713} C_VEL
LIN {X 0,Y 496.655,Z 413.994,A -85,B 0,C 180,E1 -6197.33,E2 -6197.33} C_VEL
LIN {X 0,Y 496.296,Z 425.688,A -85,B 0,C 180,E1 -6198.15,E2 -6198.15} C_VEL
LIN {X 0,Y 495.966,Z 436.26,A -85,B 0,C 180,E1 -6199.074,E2 -6199.074} C_VEL
LIN {X 0,Y 495.666,Z 444.893,A -85,B 0,C 180,E1 -6199.997,E2 -6199.997} C_VEL
LIN {X 0,Y 495.422,Z 454.239,A -85,B 0,C 180,E1 -6201.227,E2 -6201.227} C_VEL
LIN {X 0,Y 495.244,Z 461.765,A -85,B 0,C 180,E1 -6202.456,E2 -6202.456} C_VEL
LIN {X 0,Y 495.107,Z 468.178,A -85,B 0,C 180,E1 -6203.775,E2 -6203.775} C_VEL
LIN {X 0,Y 495.036,Z 473.168,A -85,B 0,C 180,E1 -6205.113,E2 -6205.113} C_VEL
LIN {X 0,Y 495.055,Z 475.567,A -85,B 0,C 180,E1 -6205.929,E2 -6205.929} C_VEL
LIN {X 0,Y 495.045,Z 477.52,A -85,B 0,C 180,E1 -6206.744,E2 -6206.744} C_VEL
LIN {X 0,Y 495.025,Z 478.986,A -85,B 0,C 180,E1 -6207.558,E2 -6207.558} C_VEL
LIN {X 0,Y 494.963,Z 480.031,A -85,B 0,C 180,E1 -6208.372,E2 -6208.372} C_VEL
LIN {X 0,Y 494.916,Z 480.674,A -85,B 0,C 180,E1 -6209.185,E2 -6209.185} C_VEL
LIN {X 0,Y 494.909,Z 480.914,A -85,B 0,C 180,E1 -6209.999,E2 -6209.999} C_VEL
LIN {X 0,Y 494.916,Z 480.703,A -85,B 0,C 180,E1 -6210.813,E2 -6210.813} C_VEL
LIN {X 0,Y 494.963,Z 480.091,A -85,B 0,C 180,E1 -6211.626,E2 -6211.626} C_VEL
LIN {X 0,Y 495.024,Z 479.079,A -85,B 0,C 180,E1 -6212.44,E2 -6212.44} C_VEL
LIN {X 0,Y 495.045,Z 477.642,A -85,B 0,C 180,E1 -6213.254,E2 -6213.254} C_VEL
LIN {X 0,Y 495.007,Z 474.632,A -85,B 0,C 180,E1 -6214.478,E2 -6214.478} C_VEL
LIN {X 0,Y 495.107,Z 470.553,A -85,B 0,C 180,E1 -6215.702,E2 -6215.702} C_VEL
LIN {X 0,Y 495.238,Z 464.253,A -85,B 0,C 180,E1 -6217.132,E2 -6217.132} C_VEL
LIN {X 0,Y 495.353,Z 457.378,A -85,B 0,C 180,E1 -6218.361,E2 -6218.361} C_VEL
LIN {X 0,Y 495.582,Z 448.816,A -85,B 0,C 180,E1 -6219.591,E2 -6219.591} C_VEL
LIN {X 0,Y 495.891,Z 439.995,A -85,B 0,C 180,E1 -6220.616,E2 -6220.616} C_VEL
LIN {X 0,Y 496.264,Z 429.141,A -85,B 0,C 180,E1 -6221.642,E2 -6221.642} C_VEL
LIN {X 0,Y 496.535,Z 418.612,A -85,B 0,C 180,E1 -6222.443,E2 -6222.443} C_VEL
LIN {X 0,Y 496.936,Z 406.177,A -85,B 0,C 180,E1 -6223.181,E2 -6223.181} C_VEL
LIN {X 0,Y 497.296,Z 393.575,A -85,B 0,C 180,E1 -6223.744,E2 -6223.744} C_VEL
LIN {X 0,Y 497.598,Z 381.39,A -85,B 0,C 180,E1 -6224.126,E2 -6224.126} C_VEL
LIN {X 0,Y 497.783,Z 364.763,A -85,B 0,C 180,E1 -6224.434,E2 -6224.434} C_VEL
LIN {X 0,Y 498.314,Z 282.403,A -85,B 0,C 180,E1 -6225.726,E2 -6225.726} C_VEL
LIN {X 0,Y 496.273,Z 268.174,A -85,B 0,C 180,E1 -6226.043,E2 -6226.043} C_VEL
LIN {X 0,Y 496.872,Z 248.233,A -85,B 0,C 180,E1 -6229.199,E2 -6229.199} C_VEL
LIN {X 0,Y 497.495,Z 230.894,A -85,B 0,C 180,E1 -6231.984,E2 -6231.984} C_VEL
LIN {X 0,Y 497.924,Z 218.864,A -85,B 0,C 180,E1 -6233.942,E2 -6233.942} C_VEL
LIN {X 0,Y 495.849,Z 207.723,A -85,B 0,C 180,E1 -6235.894,E2 -6235.894} C_VEL
LIN {X 0,Y 495.766,Z 207.729,A -85,B 0,C 180,E1 -6238.814,E2 -6238.814} C_VEL
LIN {X 0,Y 495.752,Z 207.733,A -85,B 0,C 180,E1 -6241.724,E2 -6241.724} C_VEL
LIN {X 0,Y 495.764,Z 207.721,A -85,B 0,C 180,E1 -6244.693,E2 -6244.693} C_VEL
LIN {X 0,Y 495.717,Z 207.738,A -85,B 0,C 180,E1 -6247.561,E2 -6247.561} C_VEL
LIN {X 0,Y 495.74,Z 207.734,A -85,B 0,C 180,E1 -6250.044,E2 -6250.044} C_VEL
LIN {X 0,Y 495.711,Z 207.731,A -85,B 0,C 180,E1 -6252.883,E2 -6252.883} C_VEL
LIN {X 0,Y 495.717,Z 207.735,A -85,B 0,C 180,E1 -6255.997,E2 -6255.997} C_VEL
LIN {X 0,Y 495.724,Z 207.731,A -85,B 0,C 180,E1 -6259.296,E2 -6259.296} C_VEL
LIN {X 0,Y 495.738,Z 207.736,A -85,B 0,C 180,E1 -6261.407,E2 -6261.407} C_VEL
LIN {X 0,Y 495.739,Z 207.721,A -85,B 0,C 180,E1 -6264.462,E2 -6264.462} C_VEL
LIN {X 0,Y 495.756,Z 207.731,A -85,B 0,C 180,E1 -6267.405,E2 -6267.405} C_VEL
LIN {X 0,Y 495.747,Z 207.72,A -85,B 0,C 180,E1 -6270.252,E2 -6270.252} C_VEL
LIN {X 0,Y 495.73,Z 207.734,A -85,B 0,C 180,E1 -6273.27,E2 -6273.27} C_VEL
LIN {X 0,Y 495.728,Z 207.73,A -85,B 0,C 180,E1 -6276.612,E2 -6276.612} C_VEL
LIN {X 0,Y 495.77,Z 207.724,A -85,B 0,C 180,E1 -6279.324,E2 -6279.324} C_VEL
LIN {X 0,Y 495.77,Z 207.725,A -85,B 0,C 180,E1 -6281.828,E2 -6281.828} C_VEL
LIN {X 0,Y 495.764,Z 207.717,A -85,B 0,C 180,E1 -6285.216,E2 -6285.216} C_VEL
LIN {X 0,Y 495.839,Z 207.72,A -85,B 0,C 180,E1 -6288.555,E2 -6288.555} C_VEL
LIN {X 0,Y 495.819,Z 207.719,A -85,B 0,C 180,E1 -6291.851,E2 -6291.851} C_VEL
LIN {X 0,Y 495.807,Z 207.712,A -85,B 0,C 180,E1 -6295.121,E2 -6295.121} C_VEL
LIN {X 0,Y 495.972,Z 207.698,A -85,B 0,C 180,E1 -6297.564,E2 -6297.564} C_VEL
LIN {X 0,Y 495.952,Z 207.698,A -85,B 0,C 180,E1 -6300.812,E2 -6300.812} C_VEL
LIN {X 0,Y 495.973,Z 207.693,A -85,B 0,C 180,E1 -6302.437,E2 -6302.437} C_VEL
LIN {X 0,Y 495.878,Z 207.711,A -85,B 0,C 180,E1 -6305.694,E2 -6305.694} C_VEL
LIN {X 0,Y 495.863,Z 207.715,A -85,B 0,C 180,E1 -6308.148,E2 -6308.148} C_VEL
LIN {X 0,Y 495.842,Z 207.71,A -85,B 0,C 180,E1 -6311.446,E2 -6311.446} C_VEL
LIN {X 0,Y 495.782,Z 207.722,A -85,B 0,C 180,E1 -6314.783,E2 -6314.783} C_VEL
LIN {X 0,Y 495.755,Z 207.723,A -85,B 0,C 180,E1 -6317.32,E2 -6317.32} C_VEL
LIN {X 0,Y 495.764,Z 207.732,A -85,B 0,C 180,E1 -6319.891,E2 -6319.891} C_VEL
LIN {X 0,Y 495.754,Z 207.725,A -85,B 0,C 180,E1 -6322.862,E2 -6322.862} C_VEL
LIN {X 0,Y 495.784,Z 207.726,A -85,B 0,C 180,E1 -6326.069,E2 -6326.069} C_VEL
LIN {X 0,Y 495.763,Z 207.725,A -85,B 0,C 180,E1 -6328.816,E2 -6328.816} C_VEL
LIN {X 0,Y 495.75,Z 207.732,A -85,B 0,C 180,E1 -6331.726,E2 -6331.726} C_VEL
LIN {X 0,Y 495.769,Z 207.724,A -85,B 0,C 180,E1 -6334.696,E2 -6334.696} C_VEL
LIN {X 0,Y 495.727,Z 207.732,A -85,B 0,C 180,E1 -6337.562,E2 -6337.562} C_VEL
LIN {X 0,Y 495.763,Z 207.732,A -85,B 0,C 180,E1 -6340.701,E2 -6340.701} C_VEL
LIN {X 0,Y 495.731,Z 207.731,A -85,B 0,C 180,E1 -6344.002,E2 -6344.002} C_VEL
LIN {X 0,Y 495.724,Z 207.736,A -85,B 0,C 180,E1 -6347.118,E2 -6347.118} C_VEL
LIN {X 0,Y 495.757,Z 207.727,A -85,B 0,C 180,E1 -6349.954,E2 -6349.954} C_VEL
LIN {X 0,Y 495.726,Z 207.737,A -85,B 0,C 180,E1 -6352.554,E2 -6352.554} C_VEL
LIN {X 0,Y 495.779,Z 207.727,A -85,B 0,C 180,E1 -6355.458,E2 -6355.458} C_VEL
LIN {X 0,Y 495.786,Z 207.764,A -85,B 0,C 180,E1 -6358.164,E2 -6358.164} C_VEL
LIN {X 0,Y 495.948,Z 216.376,A -85,B 0,C 180,E1 -6359.258,E2 -6359.258} C_VEL
LIN {X 0,Y 495.808,Z 219.334,A -85,B 0,C 180,E1 -6359.549,E2 -6359.549} C_VEL
LIN {X 0,Y 495.065,Z 224.58,A -85,B 0,C 180,E1 -6359.843,E2 -6359.843} C_VEL
LIN {X 0,Y 494,Z 230.269,A -85,B 0,C 180,E1 -6360.006,E2 -6360.006} C_VEL
LIN {X 0,Y 492.435,Z 238.431,A -85,B 0,C 180,E1 -6360.092,E2 -6360.092} C_VEL
LIN {X 0,Y 491.789,Z 246.688,A -85,B 0,C 180,E1 -6360.193,E2 -6360.193} C_VEL
LIN {X 0,Y 491.146,Z 332.352,A -85,B 0,C 180,E1 -6361.474,E2 -6361.474} C_VEL
LIN {X 0,Y 490.94,Z 344.802,A -85,B 0,C 180,E1 -6361.81,E2 -6361.81} C_VEL
LIN {X 0,Y 490.66,Z 357.386,A -85,B 0,C 180,E1 -6362.322,E2 -6362.322} C_VEL
LIN {X 0,Y 490.32,Z 370.332,A -85,B 0,C 180,E1 -6363.046,E2 -6363.046} C_VEL
LIN {X 0,Y 489.888,Z 381.113,A -85,B 0,C 180,E1 -6363.824,E2 -6363.824} C_VEL
LIN {X 0,Y 489.469,Z 391.507,A -85,B 0,C 180,E1 -6364.768,E2 -6364.768} C_VEL
LIN {X 0,Y 489.092,Z 400.966,A -85,B 0,C 180,E1 -6365.826,E2 -6365.826} C_VEL
LIN {X 0,Y 488.784,Z 409.222,A -85,B 0,C 180,E1 -6366.961,E2 -6366.961} C_VEL
LIN {X 0,Y 488.446,Z 416.79,A -85,B 0,C 180,E1 -6368.254,E2 -6368.254} C_VEL
LIN {X 0,Y 488.286,Z 421.861,A -85,B 0,C 180,E1 -6369.32,E2 -6369.32} C_VEL
LIN {X 0,Y 488.108,Z 426.947,A -85,B 0,C 180,E1 -6370.662,E2 -6370.662} C_VEL
LIN {X 0,Y 488.048,Z 430.459,A -85,B 0,C 180,E1 -6371.883,E2 -6371.883} C_VEL
LIN {X 0,Y 487.892,Z 433.274,A -85,B 0,C 180,E1 -6373.257,E2 -6373.257} C_VEL
LIN {X 0,Y 487.864,Z 435.105,A -85,B 0,C 180,E1 -6374.838,E2 -6374.838} C_VEL
LIN {X 0,Y 487.845,Z 435.495,A -85,B 0,C 180,E1 -6375.825,E2 -6375.825} C_VEL
LIN {X 0,Y 487.857,Z 435.409,A -85,B 0,C 180,E1 -6376.675,E2 -6376.675} C_VEL
LIN {X 0,Y 487.861,Z 434.872,A -85,B 0,C 180,E1 -6377.522,E2 -6377.522} C_VEL
LIN {X 0,Y 487.93,Z 433.928,A -85,B 0,C 180,E1 -6378.367,E2 -6378.367} C_VEL
LIN {X 0,Y 487.948,Z 432.593,A -85,B 0,C 180,E1 -6379.209,E2 -6379.209} C_VEL
LIN {X 0,Y 488.009,Z 429.755,A -85,B 0,C 180,E1 -6380.468,E2 -6380.468} C_VEL
LIN {X 0,Y 488.167,Z 425.88,A -85,B 0,C 180,E1 -6381.723,E2 -6381.723} C_VEL
LIN {X 0,Y 488.348,Z 419.703,A -85,B 0,C 180,E1 -6383.224,E2 -6383.224} C_VEL
LIN {X 0,Y 488.566,Z 413.381,A -85,B 0,C 180,E1 -6384.429,E2 -6384.429} C_VEL
LIN {X 0,Y 488.886,Z 405.298,A -85,B 0,C 180,E1 -6385.673,E2 -6385.673} C_VEL
LIN {X 0,Y 489.193,Z 397.002,A -85,B 0,C 180,E1 -6386.707,E2 -6386.707} C_VEL
LIN {X 0,Y 489.559,Z 386.863,A -85,B 0,C 180,E1 -6387.738,E2 -6387.738} C_VEL
LIN {X 0,Y 490.012,Z 376.843,A -85,B 0,C 180,E1 -6388.563,E2 -6388.563} C_VEL
LIN {X 0,Y 490.36,Z 365.946,A -85,B 0,C 180,E1 -6389.282,E2 -6389.282} C_VEL
LIN {X 0,Y 490.665,Z 353.754,A -85,B 0,C 180,E1 -6389.898,E2 -6389.898} C_VEL
LIN {X 0,Y 490.98,Z 341.116,A -85,B 0,C 180,E1 -6390.36,E2 -6390.36} C_VEL
LIN {X 0,Y 491.168,Z 327.772,A -85,B 0,C 180,E1 -6390.667,E2 -6390.667} C_VEL
LIN {X 0,Y 491.739,Z 237.2,A -85,B 0,C 180,E1 -6391.997,E2 -6391.997} C_VEL
LIN {X 0,Y 488.991,Z 222.077,A -85,B 0,C 180,E1 -6392.318,E2 -6392.318} C_VEL
LIN {X 0,Y 488.709,Z 208.613,A -85,B 0,C 180,E1 -6394.047,E2 -6394.047} C_VEL
LIN {X 0,Y 488.813,Z 208.595,A -85,B 0,C 180,E1 -6396.606,E2 -6396.606} C_VEL
LIN {X 0,Y 488.777,Z 208.604,A -85,B 0,C 180,E1 -6399.101,E2 -6399.101} C_VEL
LIN {X 0,Y 488.796,Z 208.597,A -85,B 0,C 180,E1 -6402.116,E2 -6402.116} C_VEL
LIN {X 0,Y 488.783,Z 208.601,A -85,B 0,C 180,E1 -6405.555,E2 -6405.555} C_VEL
LIN {X 0,Y 488.753,Z 208.603,A -85,B 0,C 180,E1 -6408.443,E2 -6408.443} C_VEL
LIN {X 0,Y 488.714,Z 208.61,A -85,B 0,C 180,E1 -6411.071,E2 -6411.071} C_VEL
LIN {X 0,Y 488.675,Z 208.612,A -85,B 0,C 180,E1 -6413.747,E2 -6413.747} C_VEL
LIN {X 0,Y 488.703,Z 208.611,A -85,B 0,C 180,E1 -6416.922,E2 -6416.922} C_VEL
